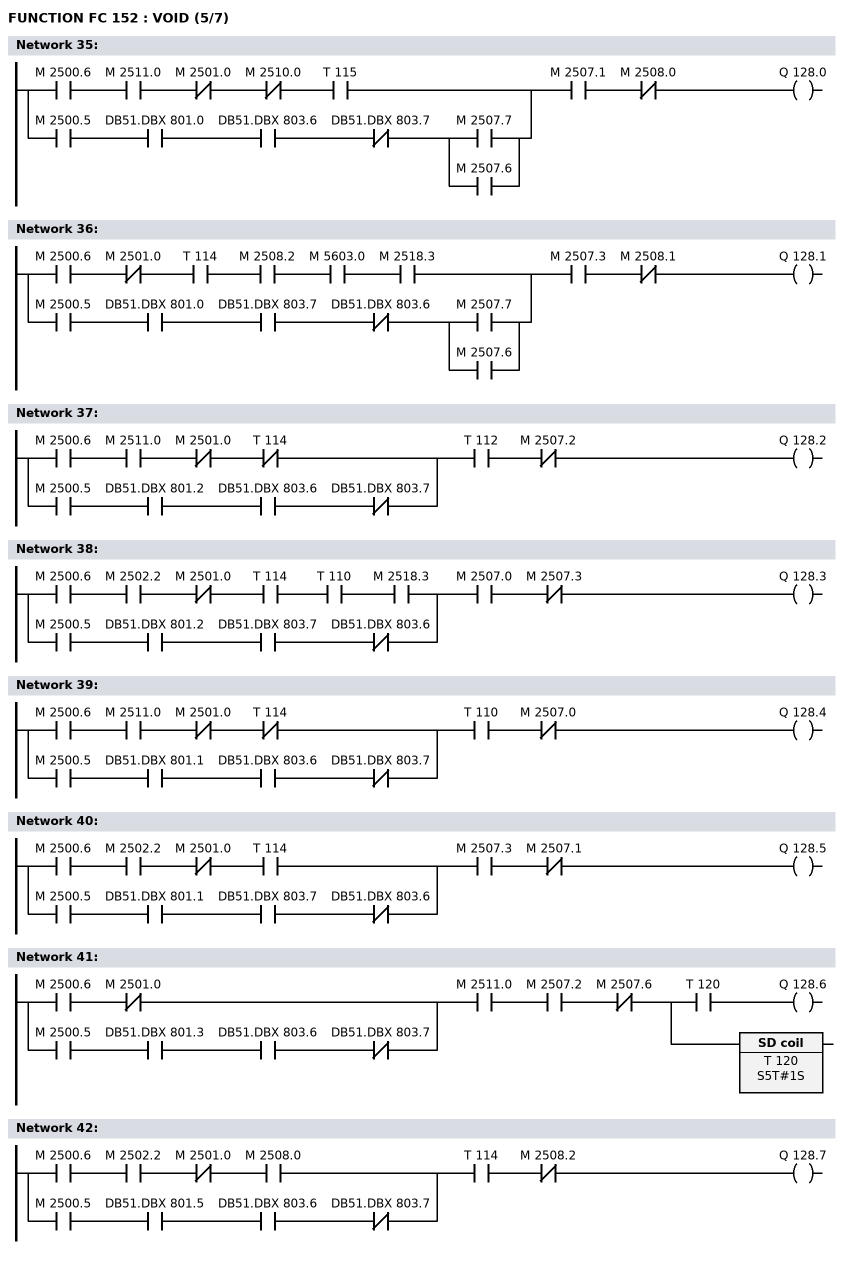

      A(    ;
      A     M   2500.6;
      A     M   2511.0;
      AN    M   2501.0;
      AN    M   2510.0;
      A     T    115;
      O     ;
      A     M   2500.5;
      A     DB51.DBX  801.0;
      A     DB51.DBX  803.6;
      AN    DB51.DBX  803.7;
      A(    ;
      O     M   2507.7;
      O     M   2507.6;
      )     ;
      )     ;
      A     M   2507.1;
      AN    M   2508.0;
      =     Q    128.0;
NETWORK
TITLE =

      A(    ;
      A     M   2500.6;
      AN    M   2501.0;
      A     T    114;
      A     M   2508.2;
      A     M   5603.0;
      A     M   2518.3;
      O     ;
      A     M   2500.5;
      A     DB51.DBX  801.0;
      A     DB51.DBX  803.7;
      AN    DB51.DBX  803.6;
      A(    ;
      O     M   2507.7;
      O     M   2507.6;
      )     ;
      )     ;
      A     M   2507.3;
      AN    M   2508.1;
      =     Q    128.1;
NETWORK
TITLE =

      A(    ;
      A     M   2500.6;
      A     M   2511.0;
      AN    M   2501.0;
      AN    T    114;
      O     ;
      A     M   2500.5;
      A     DB51.DBX  801.2;
      A     DB51.DBX  803.6;
      AN    DB51.DBX  803.7;
      )     ;
      A     T    112;
      AN    M   2507.2;
      =     Q    128.2;
NETWORK
TITLE =

      A(    ;
      A     M   2500.6;
      A     M   2502.2;
      AN    M   2501.0;
      A     T    114;
      A     T    110;
      A     M   2518.3;
      O     ;
      A     M   2500.5;
      A     DB51.DBX  801.2;
      A     DB51.DBX  803.7;
      AN    DB51.DBX  803.6;
      )     ;
      A     M   2507.0;
      AN    M   2507.3;
      =     Q    128.3;
NETWORK
TITLE =

      A(    ;
      A     M   2500.6;
      A     M   2511.0;
      AN    M   2501.0;
      AN    T    114;
      O     ;
      A     M   2500.5;
      A     DB51.DBX  801.1;
      A     DB51.DBX  803.6;
      AN    DB51.DBX  803.7;
      )     ;
      A     T    110;
      AN    M   2507.0;
      =     Q    128.4;
NETWORK
TITLE =

      A(    ;
      A     M   2500.6;
      A     M   2502.2;
      AN    M   2501.0;
      A     T    114;
      O     ;
      A     M   2500.5;
      A     DB51.DBX  801.1;
      A     DB51.DBX  803.7;
      AN    DB51.DBX  803.6;
      )     ;
      A     M   2507.3;
      AN    M   2507.1;
      =     Q    128.5;
NETWORK
TITLE =

      A(    ;
      A     M   2500.6;
      AN    M   2501.0;
      O     ;
      A     M   2500.5;
      A     DB51.DBX  801.3;
      A     DB51.DBX  803.6;
      AN    DB51.DBX  803.7;
      )     ;
      A     M   2511.0;
      A     M   2507.2;
      AN    M   2507.6;
      =     L      0.0;
      A     L      0.0;
      A     T    120;
      =     Q    128.6;
      A     L      0.0;
      BLD   102;
      L     S5T#1S;
      SD    T    120;
NETWORK
TITLE =

      A(    ;
      A     M   2500.6;
      A     M   2502.2;
      AN    M   2501.0;
      A     M   2508.0;
      O     ;
      A     M   2500.5;
      A     DB51.DBX  801.5;
      A     DB51.DBX  803.6;
      AN    DB51.DBX  803.7;
      )     ;
      A     T    114;
      AN    M   2508.2;
      =     Q    128.7;
NETWORK
TITLE =
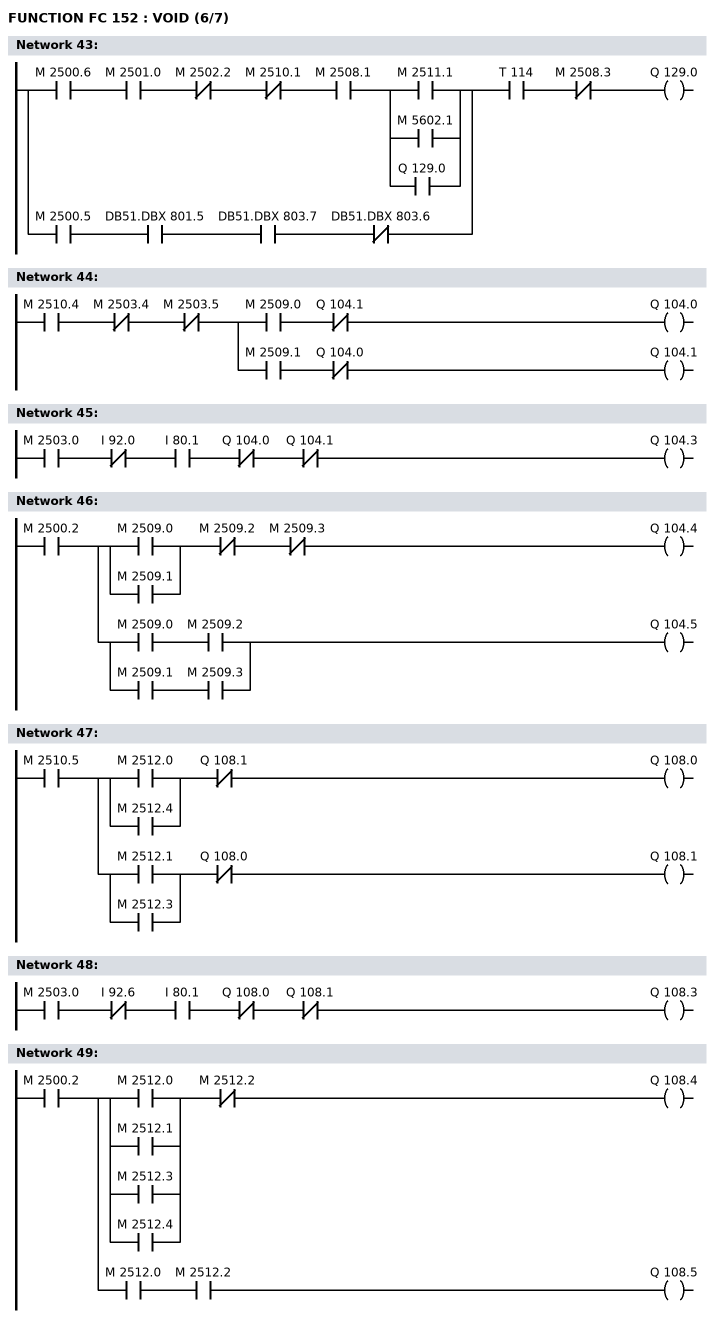

      A(    ;
      A     M   2500.6;
      A     M   2501.0;
      AN    M   2502.2;
      AN    M   2510.1;
      A     M   2508.1;
      A(    ;
      O     M   2511.1;
      O     M   5602.1;
      O     Q    129.0;
      )     ;
      O     ;
      A     M   2500.5;
      A     DB51.DBX  801.5;
      A     DB51.DBX  803.7;
      AN    DB51.DBX  803.6;
      )     ;
      A     T    114;
      AN    M   2508.3;
      =     Q    129.0;
NETWORK
TITLE =

      A     M   2510.4;
      AN    M   2503.4;
      AN    M   2503.5;
      =     L      0.0;
      A     L      0.0;
      A     M   2509.0;
      AN    Q    104.1;
      =     Q    104.0;
      A     L      0.0;
      A     M   2509.1;
      AN    Q    104.0;
      =     Q    104.1;
NETWORK
TITLE =

      A     M   2503.0;
      AN    I     92.0;
      A     I     80.1;
      AN    Q    104.0;
      AN    Q    104.1;
      =     Q    104.3;
NETWORK
TITLE =

      A     M   2500.2;
      =     L      0.0;
      A     L      0.0;
      A(    ;
      O     M   2509.0;
      O     M   2509.1;
      )     ;
      AN    M   2509.2;
      AN    M   2509.3;
      =     Q    104.4;
      A     L      0.0;
      A(    ;
      A     M   2509.0;
      A     M   2509.2;
      O     ;
      A     M   2509.1;
      A     M   2509.3;
      )     ;
      =     Q    104.5;
NETWORK
TITLE =

      A     M   2510.5;
      =     L      0.0;
      A     L      0.0;
      A(    ;
      O     M   2512.0;
      O     M   2512.4;
      )     ;
      AN    Q    108.1;
      =     Q    108.0;
      A     L      0.0;
      A(    ;
      O     M   2512.1;
      O     M   2512.3;
      )     ;
      AN    Q    108.0;
      =     Q    108.1;
NETWORK
TITLE =

      A     M   2503.0;
      AN    I     92.6;
      A     I     80.1;
      AN    Q    108.0;
      AN    Q    108.1;
      =     Q    108.3;
NETWORK
TITLE =

      A     M   2500.2;
      =     L      0.0;
      A     L      0.0;
      A(    ;
      O     M   2512.0;
      O     M   2512.1;
      O     M   2512.3;
      O     M   2512.4;
      )     ;
      AN    M   2512.2;
      =     Q    108.4;
      A     L      0.0;
      A     M   2512.0;
      A     M   2512.2;
      =     Q    108.5;
NETWORK
TITLE =
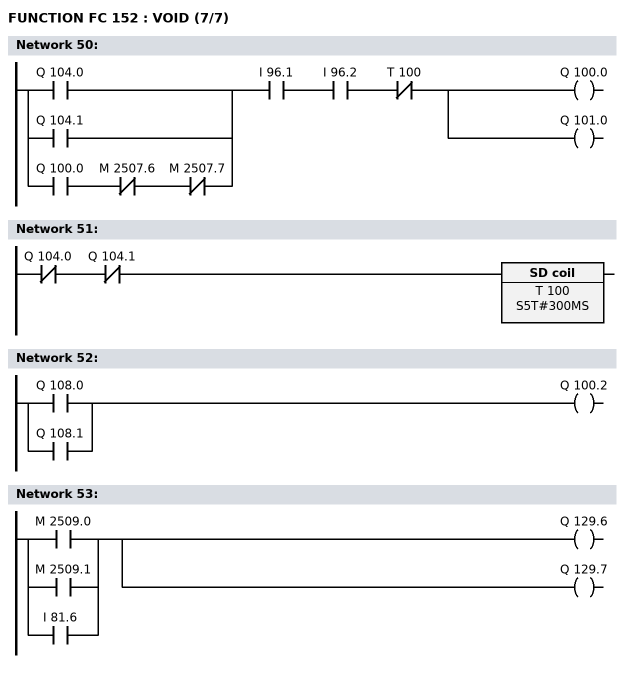

      A(    ;
      O     Q    104.0;
      O     Q    104.1;
      O     ;
      A     Q    100.0;
      AN    M   2507.6;
      AN    M   2507.7;
      )     ;
      A     I     96.1;
      A     I     96.2;
      AN    T    100;
      =     Q    100.0;
      =     Q    101.0;
NETWORK
TITLE =

      AN    Q    104.0;
      AN    Q    104.1;
      L     S5T#300MS;
      SD    T    100;
NETWORK
TITLE =

      O     Q    108.0;
      O     Q    108.1;
      =     Q    100.2;
NETWORK
TITLE =

      O     M   2509.0;
      O     M   2509.1;
      O     I     81.6;
      =     Q    129.6;
      =     Q    129.7;
END_FUNCTION

FUNCTION FC 159 : VOID
TITLE =
VERSION : 0.1

BEGIN
NETWORK
TITLE =
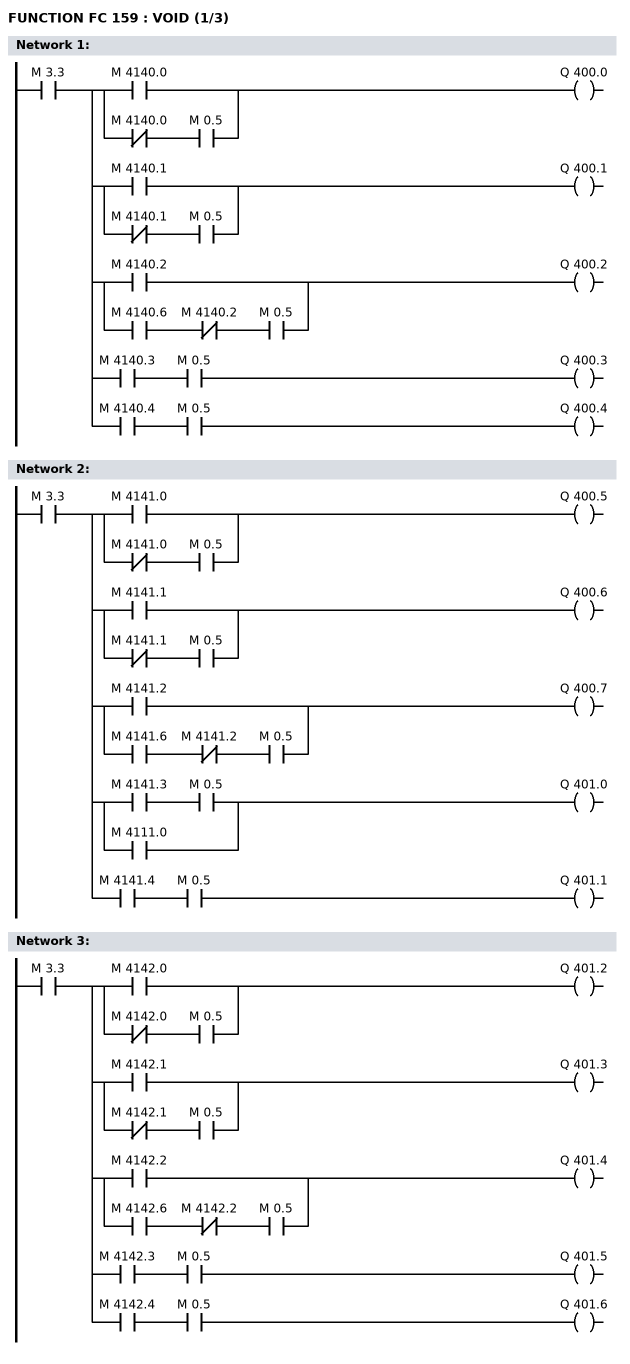

      A     M      3.3;
      =     L      0.0;
      A     L      0.0;
      A(    ;
      O     M   4140.0;
      O     ;
      AN    M   4140.0;
      A     M      0.5;
      )     ;
      =     Q    400.0;
      A     L      0.0;
      A(    ;
      O     M   4140.1;
      O     ;
      AN    M   4140.1;
      A     M      0.5;
      )     ;
      =     Q    400.1;
      A     L      0.0;
      A(    ;
      O     M   4140.2;
      O     ;
      A     M   4140.6;
      AN    M   4140.2;
      A     M      0.5;
      )     ;
      =     Q    400.2;
      A     L      0.0;
      A     M   4140.3;
      A     M      0.5;
      =     Q    400.3;
      A     L      0.0;
      A     M   4140.4;
      A     M      0.5;
      =     Q    400.4;
NETWORK
TITLE =

      A     M      3.3;
      =     L      0.0;
      A     L      0.0;
      A(    ;
      O     M   4141.0;
      O     ;
      AN    M   4141.0;
      A     M      0.5;
      )     ;
      =     Q    400.5;
      A     L      0.0;
      A(    ;
      O     M   4141.1;
      O     ;
      AN    M   4141.1;
      A     M      0.5;
      )     ;
      =     Q    400.6;
      A     L      0.0;
      A(    ;
      O     M   4141.2;
      O     ;
      A     M   4141.6;
      AN    M   4141.2;
      A     M      0.5;
      )     ;
      =     Q    400.7;
      A     L      0.0;
      A(    ;
      A     M   4141.3;
      A     M      0.5;
      O     M   4111.0;
      )     ;
      =     Q    401.0;
      A     L      0.0;
      A     M   4141.4;
      A     M      0.5;
      =     Q    401.1;
NETWORK
TITLE =

      A     M      3.3;
      =     L      0.0;
      A     L      0.0;
      A(    ;
      O     M   4142.0;
      O     ;
      AN    M   4142.0;
      A     M      0.5;
      )     ;
      =     Q    401.2;
      A     L      0.0;
      A(    ;
      O     M   4142.1;
      O     ;
      AN    M   4142.1;
      A     M      0.5;
      )     ;
      =     Q    401.3;
      A     L      0.0;
      A(    ;
      O     M   4142.2;
      O     ;
      A     M   4142.6;
      AN    M   4142.2;
      A     M      0.5;
      )     ;
      =     Q    401.4;
      A     L      0.0;
      A     M   4142.3;
      A     M      0.5;
      =     Q    401.5;
      A     L      0.0;
      A     M   4142.4;
      A     M      0.5;
      =     Q    401.6;
NETWORK
TITLE =
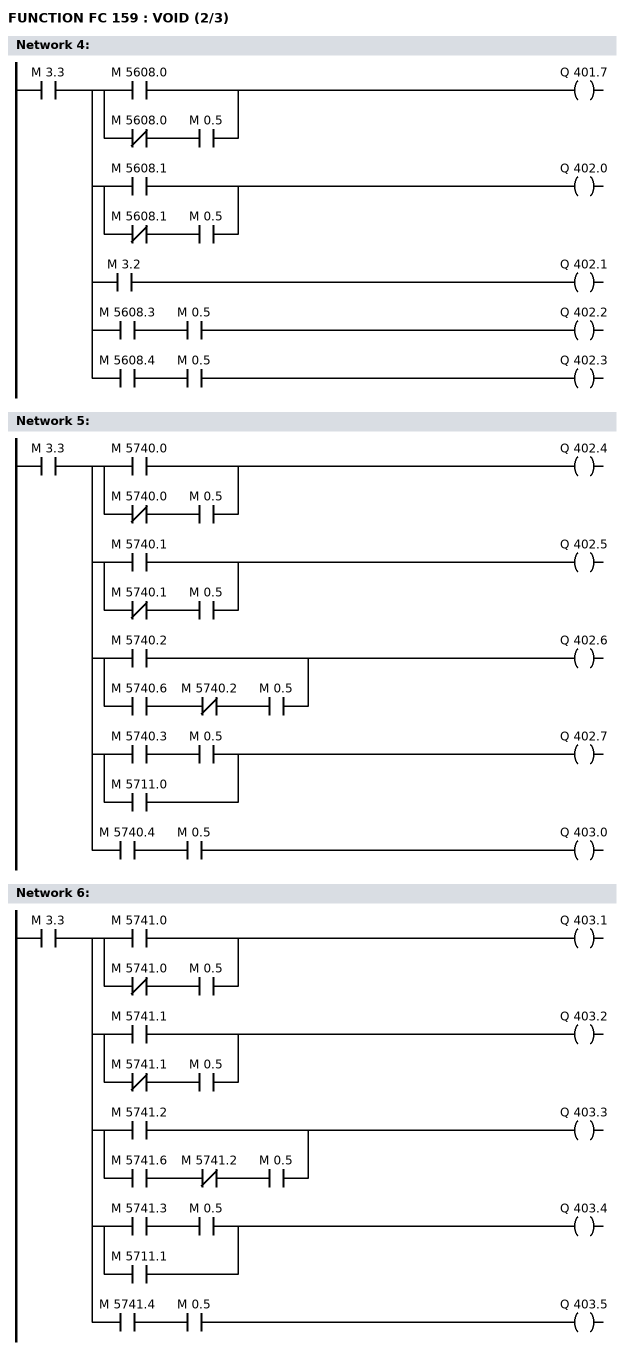

      A     M      3.3;
      =     L      0.0;
      A     L      0.0;
      A(    ;
      O     M   5608.0;
      O     ;
      AN    M   5608.0;
      A     M      0.5;
      )     ;
      =     Q    401.7;
      A     L      0.0;
      A(    ;
      O     M   5608.1;
      O     ;
      AN    M   5608.1;
      A     M      0.5;
      )     ;
      =     Q    402.0;
      A     L      0.0;
      A     M      3.2;
      =     Q    402.1;
      A     L      0.0;
      A     M   5608.3;
      A     M      0.5;
      =     Q    402.2;
      A     L      0.0;
      A     M   5608.4;
      A     M      0.5;
      =     Q    402.3;
NETWORK
TITLE =

      A     M      3.3;
      =     L      0.0;
      A     L      0.0;
      A(    ;
      O     M   5740.0;
      O     ;
      AN    M   5740.0;
      A     M      0.5;
      )     ;
      =     Q    402.4;
      A     L      0.0;
      A(    ;
      O     M   5740.1;
      O     ;
      AN    M   5740.1;
      A     M      0.5;
      )     ;
      =     Q    402.5;
      A     L      0.0;
      A(    ;
      O     M   5740.2;
      O     ;
      A     M   5740.6;
      AN    M   5740.2;
      A     M      0.5;
      )     ;
      =     Q    402.6;
      A     L      0.0;
      A(    ;
      A     M   5740.3;
      A     M      0.5;
      O     M   5711.0;
      )     ;
      =     Q    402.7;
      A     L      0.0;
      A     M   5740.4;
      A     M      0.5;
      =     Q    403.0;
NETWORK
TITLE =

      A     M      3.3;
      =     L      0.0;
      A     L      0.0;
      A(    ;
      O     M   5741.0;
      O     ;
      AN    M   5741.0;
      A     M      0.5;
      )     ;
      =     Q    403.1;
      A     L      0.0;
      A(    ;
      O     M   5741.1;
      O     ;
      AN    M   5741.1;
      A     M      0.5;
      )     ;
      =     Q    403.2;
      A     L      0.0;
      A(    ;
      O     M   5741.2;
      O     ;
      A     M   5741.6;
      AN    M   5741.2;
      A     M      0.5;
      )     ;
      =     Q    403.3;
      A     L      0.0;
      A(    ;
      A     M   5741.3;
      A     M      0.5;
      O     M   5711.1;
      )     ;
      =     Q    403.4;
      A     L      0.0;
      A     M   5741.4;
      A     M      0.5;
      =     Q    403.5;
NETWORK
TITLE =
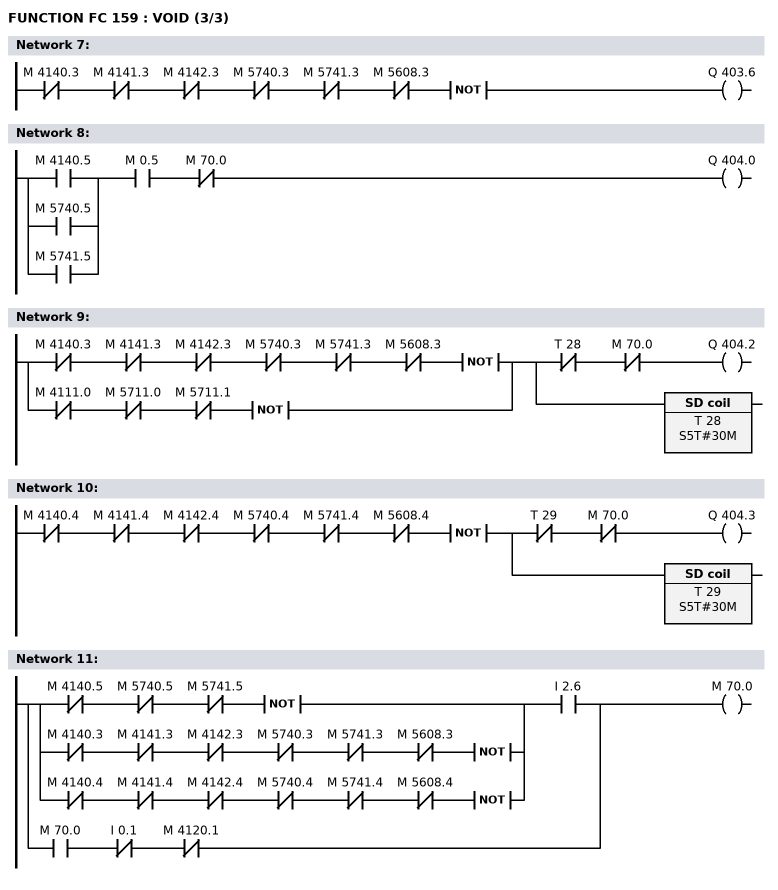

      AN    M   4140.3;
      AN    M   4141.3;
      AN    M   4142.3;
      AN    M   5740.3;
      AN    M   5741.3;
      AN    M   5608.3;
      NOT   ;
      =     Q    403.6;
NETWORK
TITLE =

      A(    ;
      O     M   4140.5;
      O     M   5740.5;
      O     M   5741.5;
      )     ;
      A     M      0.5;
      AN    M     70.0;
      =     Q    404.0;
NETWORK
TITLE =

      AN    M   4140.3;
      AN    M   4141.3;
      AN    M   4142.3;
      AN    M   5740.3;
      AN    M   5741.3;
      AN    M   5608.3;
      NOT   ;
      O(    ;
      AN    M   4111.0;
      AN    M   5711.0;
      AN    M   5711.1;
      NOT   ;
      )     ;
      =     L      0.0;
      A     L      0.0;
      AN    T     28;
      AN    M     70.0;
      =     Q    404.2;
      A     L      0.0;
      BLD   102;
      L     S5T#30M;
      SD    T     28;
NETWORK
TITLE =

      AN    M   4140.4;
      AN    M   4141.4;
      AN    M   4142.4;
      AN    M   5740.4;
      AN    M   5741.4;
      AN    M   5608.4;
      NOT   ;
      =     L      0.0;
      A     L      0.0;
      AN    T     29;
      AN    M     70.0;
      =     Q    404.3;
      A     L      0.0;
      BLD   102;
      L     S5T#30M;
      SD    T     29;
NETWORK
TITLE =

      A(    ;
      AN    M   4140.5;
      AN    M   5740.5;
      AN    M   5741.5;
      NOT   ;
      O(    ;
      AN    M   4140.3;
      AN    M   4141.3;
      AN    M   4142.3;
      AN    M   5740.3;
      AN    M   5741.3;
      AN    M   5608.3;
      NOT   ;
      )     ;
      O(    ;
      AN    M   4140.4;
      AN    M   4141.4;
      AN    M   4142.4;
      AN    M   5740.4;
      AN    M   5741.4;
      AN    M   5608.4;
      NOT   ;
      )     ;
      )     ;
      A     I      2.6;
      O     ;
      A     M     70.0;
      AN    I      0.1;
      AN    M   4120.1;
      =     M     70.0;
END_FUNCTION

FUNCTION FC 324 : VOID
TITLE =
VERSION : 0.1

BEGIN
NETWORK
TITLE =DP DIAGNOSTIC FOR DP MASTER SYSTEM(1)

      AN    OV;
      =     L      0.0;
      BLD   103;
      A     OV;
      =     L      0.1;
      BLD   103;
      CALL FC   325 (
           CHECK_ACTIV              := L      0.0,
           EXTERNAL_DP_INTERFACE    := L      0.1,
           DP_MASTERSYSTEM          := 1,
           DATA_FIELD               := P#DB325.DBX0.0 BYTE 50,
           SUM_SLAVES_DIAG          := DB325.DBW   82,
           LIST_SLAVES_NOT_PRESENT  := P#DB325.DBX 50.0 DWORD 4,
           LIST_SLAVES_ERROR        := P#DB325.DBX 66.0 DWORD 4,
           RETVAL                   := DB325.DBW   84,
           BUSY                     := DB325.DBX   90.0);
      NOP   0;
NETWORK
TITLE =705R1
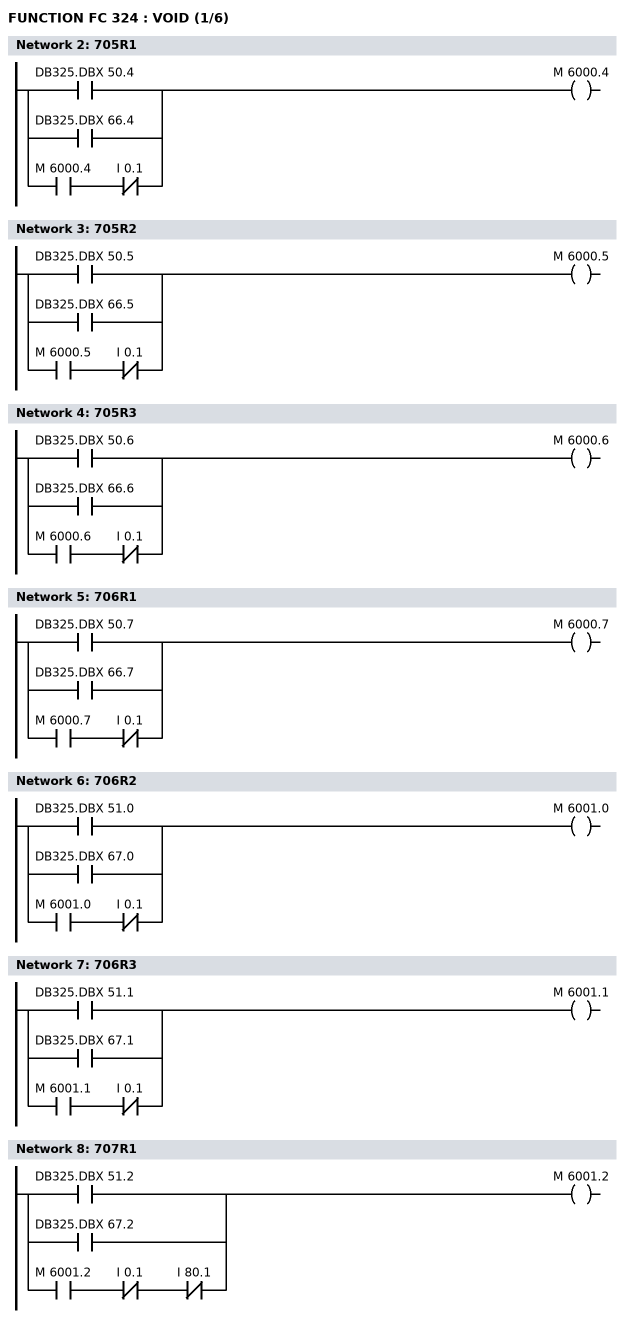

      O     DB325.DBX   50.4;
      O     DB325.DBX   66.4;
      O     ;
      A     M   6000.4;
      AN    I      0.1;
      =     M   6000.4;
NETWORK
TITLE =705R2

      O     DB325.DBX   50.5;
      O     DB325.DBX   66.5;
      O     ;
      A     M   6000.5;
      AN    I      0.1;
      =     M   6000.5;
NETWORK
TITLE =705R3

      O     DB325.DBX   50.6;
      O     DB325.DBX   66.6;
      O     ;
      A     M   6000.6;
      AN    I      0.1;
      =     M   6000.6;
NETWORK
TITLE =706R1

      O     DB325.DBX   50.7;
      O     DB325.DBX   66.7;
      O     ;
      A     M   6000.7;
      AN    I      0.1;
      =     M   6000.7;
NETWORK
TITLE =706R2

      O     DB325.DBX   51.0;
      O     DB325.DBX   67.0;
      O     ;
      A     M   6001.0;
      AN    I      0.1;
      =     M   6001.0;
NETWORK
TITLE =706R3

      O     DB325.DBX   51.1;
      O     DB325.DBX   67.1;
      O     ;
      A     M   6001.1;
      AN    I      0.1;
      =     M   6001.1;
NETWORK
TITLE =707R1

      O     DB325.DBX   51.2;
      O     DB325.DBX   67.2;
      O     ;
      A     M   6001.2;
      AN    I      0.1;
      AN    I     80.1;
      =     M   6001.2;
NETWORK
TITLE =707R2
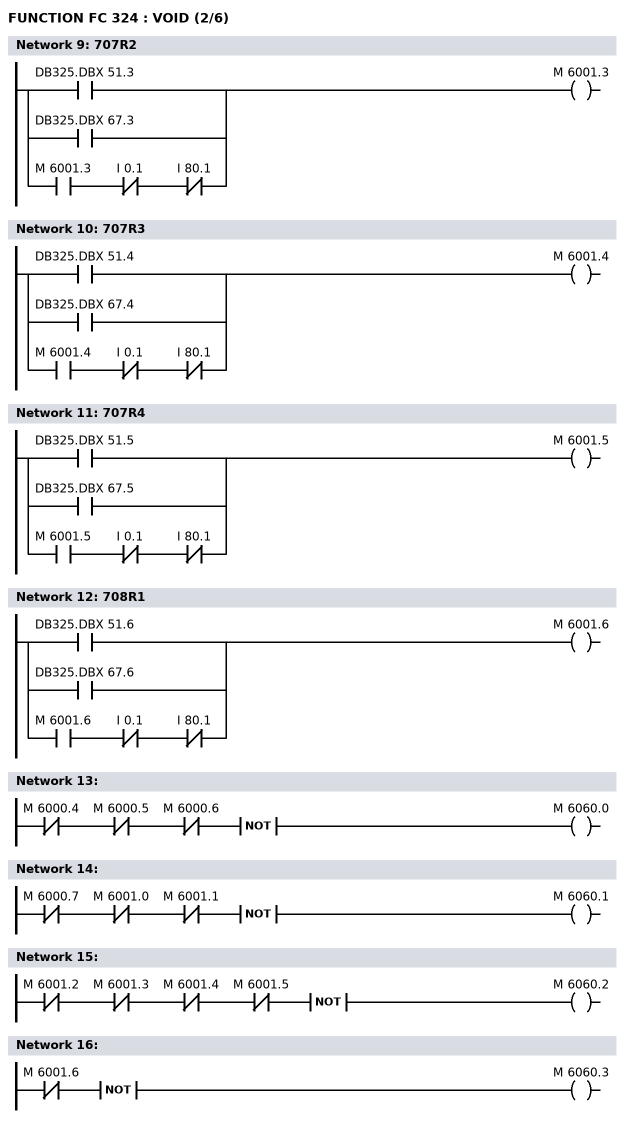

      O     DB325.DBX   51.3;
      O     DB325.DBX   67.3;
      O     ;
      A     M   6001.3;
      AN    I      0.1;
      AN    I     80.1;
      =     M   6001.3;
NETWORK
TITLE =707R3

      O     DB325.DBX   51.4;
      O     DB325.DBX   67.4;
      O     ;
      A     M   6001.4;
      AN    I      0.1;
      AN    I     80.1;
      =     M   6001.4;
NETWORK
TITLE =707R4

      O     DB325.DBX   51.5;
      O     DB325.DBX   67.5;
      O     ;
      A     M   6001.5;
      AN    I      0.1;
      AN    I     80.1;
      =     M   6001.5;
NETWORK
TITLE =708R1

      O     DB325.DBX   51.6;
      O     DB325.DBX   67.6;
      O     ;
      A     M   6001.6;
      AN    I      0.1;
      AN    I     80.1;
      =     M   6001.6;
NETWORK
TITLE =

      AN    M   6000.4;
      AN    M   6000.5;
      AN    M   6000.6;
      NOT   ;
      =     M   6060.0;
NETWORK
TITLE =

      AN    M   6000.7;
      AN    M   6001.0;
      AN    M   6001.1;
      NOT   ;
      =     M   6060.1;
NETWORK
TITLE =

      AN    M   6001.2;
      AN    M   6001.3;
      AN    M   6001.4;
      AN    M   6001.5;
      NOT   ;
      =     M   6060.2;
NETWORK
TITLE =

      AN    M   6001.6;
      NOT   ;
      =     M   6060.3;
NETWORK
TITLE =
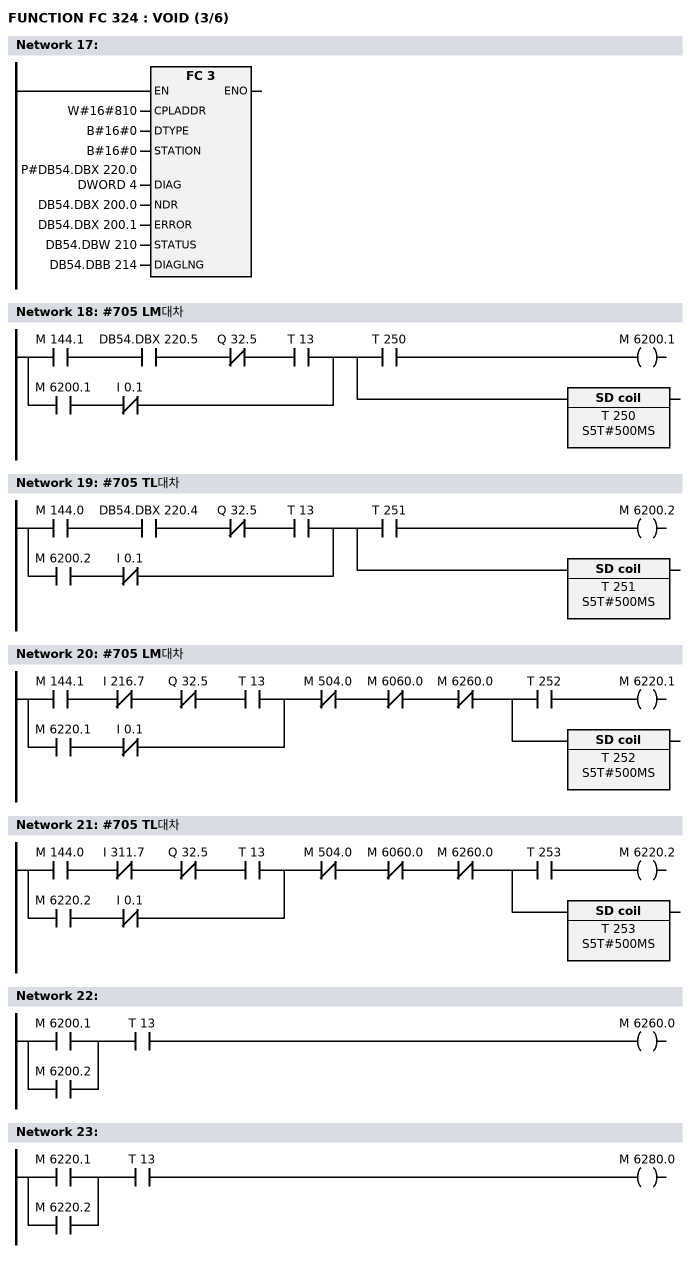

      CALL FC     3 (
           CPLADDR                  := W#16#810,
           DTYPE                    := B#16#0,
           STATION                  := B#16#0,
           DIAG                     := P#DB54.DBX 220.0 DWORD 4,
           NDR                      := DB54.DBX  200.0,
           ERROR                    := DB54.DBX  200.1,
           STATUS                   := DB54.DBW  210,
           DIAGLNG                  := DB54.DBB  214);
      NOP   0;
NETWORK
TITLE =#705 LM대차

      A     M    144.1;
      A     DB54.DBX  220.5;
      AN    Q     32.5;
      A     T     13;
      O     ;
      A     M   6200.1;
      AN    I      0.1;
      =     L      0.0;
      A     L      0.0;
      A     T    250;
      =     M   6200.1;
      A     L      0.0;
      BLD   102;
      L     S5T#500MS;
      SD    T    250;
NETWORK
TITLE =#705 TL대차

      A     M    144.0;
      A     DB54.DBX  220.4;
      AN    Q     32.5;
      A     T     13;
      O     ;
      A     M   6200.2;
      AN    I      0.1;
      =     L      0.0;
      A     L      0.0;
      A     T    251;
      =     M   6200.2;
      A     L      0.0;
      BLD   102;
      L     S5T#500MS;
      SD    T    251;
NETWORK
TITLE =#705 LM대차

      A(    ;
      A     M    144.1;
      AN    I    216.7;
      AN    Q     32.5;
      A     T     13;
      O     ;
      A     M   6220.1;
      AN    I      0.1;
      )     ;
      AN    M    504.0;
      AN    M   6060.0;
      AN    M   6260.0;
      =     L      0.0;
      A     L      0.0;
      A     T    252;
      =     M   6220.1;
      A     L      0.0;
      BLD   102;
      L     S5T#500MS;
      SD    T    252;
NETWORK
TITLE =#705 TL대차

      A(    ;
      A     M    144.0;
      AN    I    311.7;
      AN    Q     32.5;
      A     T     13;
      O     ;
      A     M   6220.2;
      AN    I      0.1;
      )     ;
      AN    M    504.0;
      AN    M   6060.0;
      AN    M   6260.0;
      =     L      0.0;
      A     L      0.0;
      A     T    253;
      =     M   6220.2;
      A     L      0.0;
      BLD   102;
      L     S5T#500MS;
      SD    T    253;
NETWORK
TITLE =

      A(    ;
      O     M   6200.1;
      O     M   6200.2;
      )     ;
      A     T     13;
      =     M   6260.0;
NETWORK
TITLE =

      A(    ;
      O     M   6220.1;
      O     M   6220.2;
      )     ;
      A     T     13;
      =     M   6280.0;
NETWORK
TITLE =
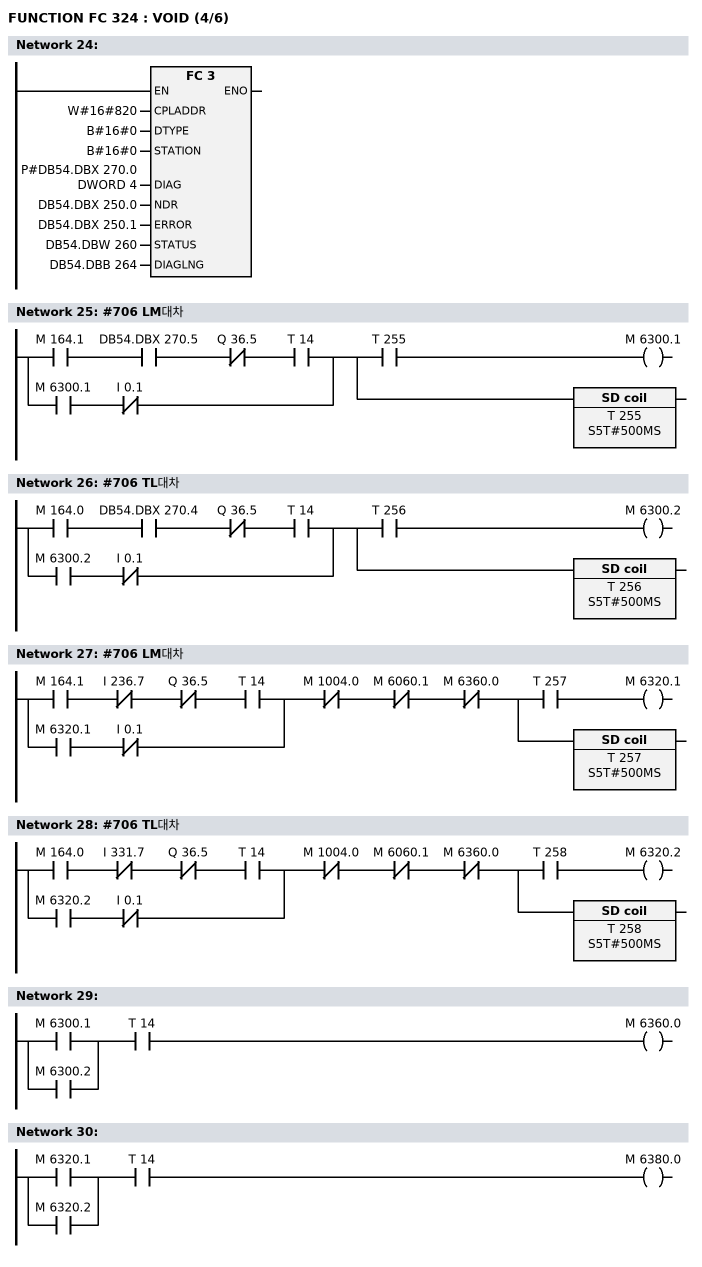

      CALL FC     3 (
           CPLADDR                  := W#16#820,
           DTYPE                    := B#16#0,
           STATION                  := B#16#0,
           DIAG                     := P#DB54.DBX 270.0 DWORD 4,
           NDR                      := DB54.DBX  250.0,
           ERROR                    := DB54.DBX  250.1,
           STATUS                   := DB54.DBW  260,
           DIAGLNG                  := DB54.DBB  264);
      NOP   0;
NETWORK
TITLE =#706 LM대차

      A     M    164.1;
      A     DB54.DBX  270.5;
      AN    Q     36.5;
      A     T     14;
      O     ;
      A     M   6300.1;
      AN    I      0.1;
      =     L      0.0;
      A     L      0.0;
      A     T    255;
      =     M   6300.1;
      A     L      0.0;
      BLD   102;
      L     S5T#500MS;
      SD    T    255;
NETWORK
TITLE =#706 TL대차

      A     M    164.0;
      A     DB54.DBX  270.4;
      AN    Q     36.5;
      A     T     14;
      O     ;
      A     M   6300.2;
      AN    I      0.1;
      =     L      0.0;
      A     L      0.0;
      A     T    256;
      =     M   6300.2;
      A     L      0.0;
      BLD   102;
      L     S5T#500MS;
      SD    T    256;
NETWORK
TITLE =#706 LM대차

      A(    ;
      A     M    164.1;
      AN    I    236.7;
      AN    Q     36.5;
      A     T     14;
      O     ;
      A     M   6320.1;
      AN    I      0.1;
      )     ;
      AN    M   1004.0;
      AN    M   6060.1;
      AN    M   6360.0;
      =     L      0.0;
      A     L      0.0;
      A     T    257;
      =     M   6320.1;
      A     L      0.0;
      BLD   102;
      L     S5T#500MS;
      SD    T    257;
NETWORK
TITLE =#706 TL대차

      A(    ;
      A     M    164.0;
      AN    I    331.7;
      AN    Q     36.5;
      A     T     14;
      O     ;
      A     M   6320.2;
      AN    I      0.1;
      )     ;
      AN    M   1004.0;
      AN    M   6060.1;
      AN    M   6360.0;
      =     L      0.0;
      A     L      0.0;
      A     T    258;
      =     M   6320.2;
      A     L      0.0;
      BLD   102;
      L     S5T#500MS;
      SD    T    258;
NETWORK
TITLE =

      A(    ;
      O     M   6300.1;
      O     M   6300.2;
      )     ;
      A     T     14;
      =     M   6360.0;
NETWORK
TITLE =

      A(    ;
      O     M   6320.1;
      O     M   6320.2;
      )     ;
      A     T     14;
      =     M   6380.0;
NETWORK
TITLE =
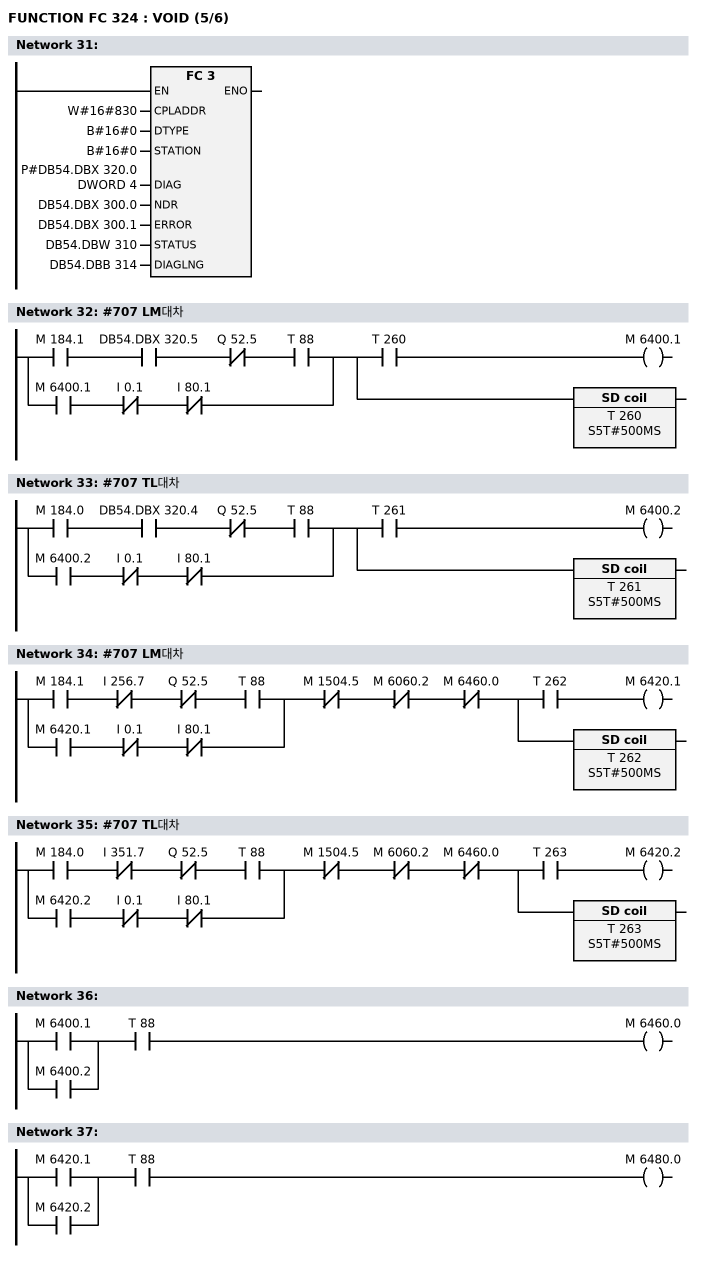

      CALL FC     3 (
           CPLADDR                  := W#16#830,
           DTYPE                    := B#16#0,
           STATION                  := B#16#0,
           DIAG                     := P#DB54.DBX 320.0 DWORD 4,
           NDR                      := DB54.DBX  300.0,
           ERROR                    := DB54.DBX  300.1,
           STATUS                   := DB54.DBW  310,
           DIAGLNG                  := DB54.DBB  314);
      NOP   0;
NETWORK
TITLE =#707 LM대차

      A     M    184.1;
      A     DB54.DBX  320.5;
      AN    Q     52.5;
      A     T     88;
      O     ;
      A     M   6400.1;
      AN    I      0.1;
      AN    I     80.1;
      =     L      0.0;
      A     L      0.0;
      A     T    260;
      =     M   6400.1;
      A     L      0.0;
      BLD   102;
      L     S5T#500MS;
      SD    T    260;
NETWORK
TITLE =#707 TL대차

      A     M    184.0;
      A     DB54.DBX  320.4;
      AN    Q     52.5;
      A     T     88;
      O     ;
      A     M   6400.2;
      AN    I      0.1;
      AN    I     80.1;
      =     L      0.0;
      A     L      0.0;
      A     T    261;
      =     M   6400.2;
      A     L      0.0;
      BLD   102;
      L     S5T#500MS;
      SD    T    261;
NETWORK
TITLE =#707 LM대차

      A(    ;
      A     M    184.1;
      AN    I    256.7;
      AN    Q     52.5;
      A     T     88;
      O     ;
      A     M   6420.1;
      AN    I      0.1;
      AN    I     80.1;
      )     ;
      AN    M   1504.5;
      AN    M   6060.2;
      AN    M   6460.0;
      =     L      0.0;
      A     L      0.0;
      A     T    262;
      =     M   6420.1;
      A     L      0.0;
      BLD   102;
      L     S5T#500MS;
      SD    T    262;
NETWORK
TITLE =#707 TL대차

      A(    ;
      A     M    184.0;
      AN    I    351.7;
      AN    Q     52.5;
      A     T     88;
      O     ;
      A     M   6420.2;
      AN    I      0.1;
      AN    I     80.1;
      )     ;
      AN    M   1504.5;
      AN    M   6060.2;
      AN    M   6460.0;
      =     L      0.0;
      A     L      0.0;
      A     T    263;
      =     M   6420.2;
      A     L      0.0;
      BLD   102;
      L     S5T#500MS;
      SD    T    263;
NETWORK
TITLE =

      A(    ;
      O     M   6400.1;
      O     M   6400.2;
      )     ;
      A     T     88;
      =     M   6460.0;
NETWORK
TITLE =

      A(    ;
      O     M   6420.1;
      O     M   6420.2;
      )     ;
      A     T     88;
      =     M   6480.0;
NETWORK
TITLE =
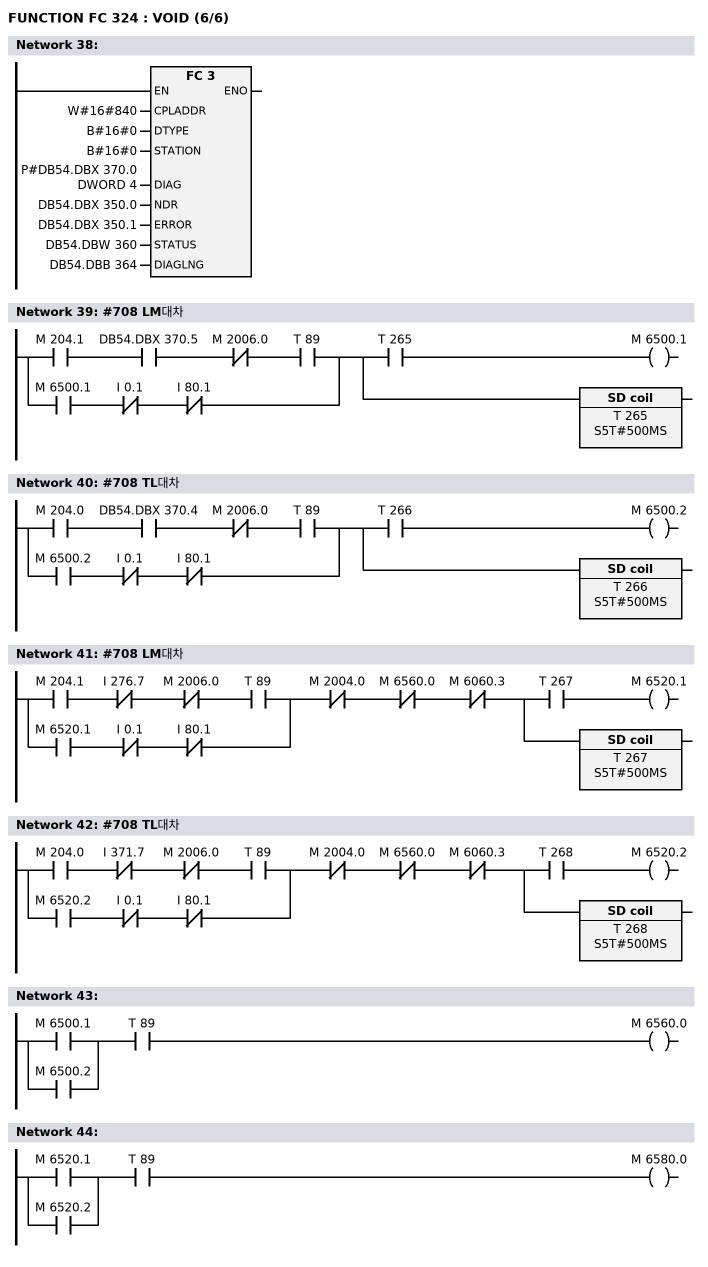

      CALL FC     3 (
           CPLADDR                  := W#16#840,
           DTYPE                    := B#16#0,
           STATION                  := B#16#0,
           DIAG                     := P#DB54.DBX 370.0 DWORD 4,
           NDR                      := DB54.DBX  350.0,
           ERROR                    := DB54.DBX  350.1,
           STATUS                   := DB54.DBW  360,
           DIAGLNG                  := DB54.DBB  364);
      NOP   0;
NETWORK
TITLE =#708 LM대차

      A     M    204.1;
      A     DB54.DBX  370.5;
      AN    M   2006.0;
      A     T     89;
      O     ;
      A     M   6500.1;
      AN    I      0.1;
      AN    I     80.1;
      =     L      0.0;
      A     L      0.0;
      A     T    265;
      =     M   6500.1;
      A     L      0.0;
      BLD   102;
      L     S5T#500MS;
      SD    T    265;
NETWORK
TITLE =#708 TL대차

      A     M    204.0;
      A     DB54.DBX  370.4;
      AN    M   2006.0;
      A     T     89;
      O     ;
      A     M   6500.2;
      AN    I      0.1;
      AN    I     80.1;
      =     L      0.0;
      A     L      0.0;
      A     T    266;
      =     M   6500.2;
      A     L      0.0;
      BLD   102;
      L     S5T#500MS;
      SD    T    266;
NETWORK
TITLE =#708 LM대차

      A(    ;
      A     M    204.1;
      AN    I    276.7;
      AN    M   2006.0;
      A     T     89;
      O     ;
      A     M   6520.1;
      AN    I      0.1;
      AN    I     80.1;
      )     ;
      AN    M   2004.0;
      AN    M   6560.0;
      AN    M   6060.3;
      =     L      0.0;
      A     L      0.0;
      A     T    267;
      =     M   6520.1;
      A     L      0.0;
      BLD   102;
      L     S5T#500MS;
      SD    T    267;
NETWORK
TITLE =#708 TL대차

      A(    ;
      A     M    204.0;
      AN    I    371.7;
      AN    M   2006.0;
      A     T     89;
      O     ;
      A     M   6520.2;
      AN    I      0.1;
      AN    I     80.1;
      )     ;
      AN    M   2004.0;
      AN    M   6560.0;
      AN    M   6060.3;
      =     L      0.0;
      A     L      0.0;
      A     T    268;
      =     M   6520.2;
      A     L      0.0;
      BLD   102;
      L     S5T#500MS;
      SD    T    268;
NETWORK
TITLE =

      A(    ;
      O     M   6500.1;
      O     M   6500.2;
      )     ;
      A     T     89;
      =     M   6560.0;
NETWORK
TITLE =

      A(    ;
      O     M   6520.1;
      O     M   6520.2;
      )     ;
      A     T     89;
      =     M   6580.0;
END_FUNCTION

FUNCTION_BLOCK FB 406
TITLE =Data Block Move Program
AUTHOR : HMC
FAMILY : Car_Type
NAME : Car_Type
VERSION : 1.0


VAR_INPUT
  FWD_Pulse : BOOL ;
  RET_Pulse : BOOL ;
  Source_DB : INT ;
  Start_Add : INT ;
  Stn_Amount : INT ;
  Byte_per_Stn : INT ;
  Cpu_Run_Pulse : BOOL ;
END_VAR
VAR_OUTPUT
  Complete : BOOL ;
END_VAR
VAR
  Operation : BOOL ;
  Mask_Arr : ARRAY  [0 .. 599 ] OF BYTE ;
  Ret : INT ;
  Data_Type : WORD ;
  Data_Length : INT ;
  Secend_Stn_Add : INT ;
  Fill_Source : WORD ;
END_VAR
VAR_TEMP
  First_Stn : ANY ;
  Mask : ANY ;
  Second_Stn : ANY ;
  Save_AR1 : DWORD ;
  Save_AR2 : DWORD ;
  Save_DB : INT ;
  Save_DI : INT ;
  First_Stn_1 : ANY ;
END_VAR
BEGIN
NETWORK
TITLE =Save adress register and DB's

      TAR1  #Save_AR1; // Save adress register 1
      TAR2  #Save_AR2; // Save adress register 2
      L     DBNO; // loads the number of the shared open data block
      T     #Save_DB;
      L     DINO; // loads the number of the opened instance data block
      T     #Save_DI;
NETWORK
TITLE =Operation Pulse

      O     #FWD_Pulse; // External ForwardOperation Signal
      O     #RET_Pulse; // External Return Operation Signal
      FP    #Operation; // Operation Pulse
      JNB   _End; // Jump to End
NETWORK
TITLE =Data Type Select In ANY Type Parameter

      A(    ; // If Source DB is Not Zero
      L     #Source_DB;
      L     0;
      <>I   ;
      )     ;
      JNB   _001; // Jump to Next Step
      L     W#16#8400; // Load "8400" _ Means "DB Area"
      T     #Data_Type; // Transfer to Data_Type
_001: NOP   0;
NETWORK
TITLE =Data Type Select In ANY Type Parameter

      A(    ; // If DB_NO is Zero
      L     #Source_DB;
      L     0;
      ==I   ;
      )     ;
      JNB   _002; // Jump to Next Step
      L     W#16#8300; // Load "8300" _ Means "Bit Memory Area"
      T     #Data_Type; // Transfer to Data_Type
_002: NOP   0;
NETWORK
TITLE =Data Length Select

      L     #Stn_Amount; // Station Amount - 1
      L     1;
      -I    ;
      L     #Byte_per_Stn; // Multi Length Per Station
      *I    ;
      T     #Data_Length; // Transfer to Data Length
NETWORK
TITLE =2nd Station Address Select

      L     #Start_Add; // Pluse Start Address And Length
      L     #Byte_per_Stn;
      +I    ;
      T     #Secend_Stn_Add; // Transfer to Second Station Address
NETWORK
TITLE =Make a "ANY" Type Data

      LAR1  P##First_Stn; // Load 1st Station Address of ANY Pointer In "AR1"

      L     B#16#10; // Load Syntax ID For S7 "10"
      T     LB [AR1,P#0.0]; // Transfer ID to the ANY Pointer

      L     B#16#2; // Load Data Type _ "2" means "BYTE"
      T     LB [AR1,P#1.0]; // Transfer Data Type to the ANY Pointer

      L     #Data_Length; // Load the Length of Source Data
      T     LW [AR1,P#2.0]; // Transfer the Numbers to the ANY Pointer

      L     #Source_DB; // Load DB Number _ "0" means don't use "DB"
      T     LW [AR1,P#4.0]; // Transfer the Numbers to the ANY Pointer

      L     #Data_Type; // Load Data Type _ "83" means "Bit Memory" Area
      T     LW [AR1,P#6.0]; //                  "84" means "DB" Area

      L     #Start_Add; // Load Start Address
      SLW   3; // Shift Left Word _ "3" Bit
      T     LW [AR1,P#8.0]; // Transfer the Address to the ANY Pointer

      LAR1  P##Mask; // Load 2nd Station Address of ANY Pointer In "AR1"

      L     B#16#10; //Load Syntax ID For S7 "10"
      T     LB [AR1,P#0.0]; //Load Syntax ID For S7 "10"

      L     B#16#2; //  Load Data Type _ "2" means "BYTE"
      T     LB [AR1,P#1.0]; // Transfer Data Type to the ANY Pointer

      L     #Data_Length; // Load the Length of Target Data
      T     LW [AR1,P#2.0]; // Transfer the Numbers to the ANY Pointer

      L     #Save_DI; // Load DB Number _ "0" means don't use "DB"
      T     LW [AR1,P#4.0]; // Transfer the Numbers to the ANY Pointer

      L     #Data_Type; // Load Data Type _ "83" means "Bit Memory" Area
      T     LW [AR1,P#6.0]; //                  "84" means "DB" Area

      L     16; //  Load Start Address
      SLW   3; // Shift Left Word _ "3" Bit
      T     LW [AR1,P#8.0]; // Transfer the Address to the ANY Pointer

NETWORK
TITLE =Make a "ANY" Type Data

      LAR1  P##Second_Stn; // Load 1st Station Address of ANY Pointer In "AR1"

      L     B#16#10; // Load Syntax ID For S7 "10"
      T     LB [AR1,P#0.0]; // Transfer ID to the ANY Pointer

      L     B#16#2; // Load Data Type _ "2" means "BYTE"
      T     LB [AR1,P#1.0]; // Transfer Data Type to the ANY Pointer

      L     #Data_Length; // Load the Length of Source Data
      T     LW [AR1,P#2.0]; // Transfer the Numbers to the ANY Pointer

      L     #Source_DB; // Load DB Number _ "0" means don't use "DB"
      T     LW [AR1,P#4.0]; // Transfer the Numbers to the ANY Pointer

      L     #Data_Type; // Load Data Type _ "83" means "Bit Memory" Area
      T     LW [AR1,P#6.0]; //                  "84" means "DB" Area

      L     #Secend_Stn_Add; // Load Second Station Address
      SLW   3; // Shift Left Word _ "3" Bit
      T     LW [AR1,P#8.0]; // Transfer the Address to the ANY Pointer
NETWORK
TITLE =Reset Car Type Transfer Complete Signal

      O     #FWD_Pulse; // External Forward Operation Signal
      O     #RET_Pulse; // External Return Operation Signal
      R     #Complete; // Reset Complete Signal
NETWORK
TITLE =Make Fill Source Data

      L     0;
      T     #Fill_Source;
NETWORK
TITLE =Fwd Block Move to Mask Area

      A     #FWD_Pulse; // External Forward Operation Signal
      AN    #Complete; // Complete Signal is False
      AN    #Cpu_Run_Pulse;
      JNB   _FWD;
      CALL SFC   20 (
           SRCBLK                   := #First_Stn,
           RET_VAL                  := #Ret,
           DSTBLK                   := #Mask);

NETWORK
TITLE =Clear Source Data Area


      CALL SFC   21 (
           IN0                      := #Fill_Source,// "Zero"
           RET_VAL                  := #Ret,
           OUT1                     := #First_Stn);// Transfer to First Station Area

NETWORK
TITLE =Fwd Block Move to Second Station Area


      CALL SFC   20 (
           SRCBLK                   := #Mask,
           RET_VAL                  := #Ret,
           DSTBLK                   := #Second_Stn);

NETWORK
TITLE =Clear Mask Data Area


      CALL SFC   21 (
           IN0                      := #Fill_Source,// "Zero"
           RET_VAL                  := #Ret,
           OUT1                     := #Mask);// Transfer to Mask Area
_FWD: NOP   0;
NETWORK
TITLE =Rev Block Move to Mask Area

      A     #RET_Pulse; // External Return Operation Signal
      AN    #Complete; // Complete Signal is False
      AN    #Cpu_Run_Pulse;
      JNB   _REV;
      CALL SFC   20 (
           SRCBLK                   := #Second_Stn,
           RET_VAL                  := #Ret,
           DSTBLK                   := #Mask);

NETWORK
TITLE =Clear Source Data Area


      CALL SFC   21 (
           IN0                      := #Fill_Source,// "Zero"
           RET_VAL                  := #Ret,
           OUT1                     := #Second_Stn);// Transfer to Second Station Area

NETWORK
TITLE =Rev Block Move to First Station Area


      CALL SFC   20 (
           SRCBLK                   := #Mask,
           RET_VAL                  := #Ret,
           DSTBLK                   := #First_Stn);

NETWORK
TITLE =Clear Mask Data Area


      CALL SFC   21 (
           IN0                      := #Fill_Source,// "Zero"
           RET_VAL                  := #Ret,
           OUT1                     := #Mask);// Transfer to Mask Area
_REV: NOP   0;
NETWORK
TITLE =Set Complete Signal

      S     #Complete;
_End: NOP   0;
END_FUNCTION_BLOCK

FUNCTION_BLOCK FB 470
TITLE =HMI Body Type Modify Variables Program
AUTHOR : HMC
FAMILY : HMI
NAME : HMI
VERSION : 1.0


VAR_INPUT
  Station : INT ;
  HMI_Disp_DB : INT ;
  HMI_Disp_Add : INT ;
  CType_DB : INT ;
  CType_Start_Add : INT ;
  Byte_per_Stn : INT ;
  M_Modify_OK : BOOL ;
  SS_CCR_On : BOOL ;
  PB_Set : BOOL ;
  PB_Reset : BOOL ;
END_VAR
VAR_OUTPUT
  LP_CCR_On : BOOL ;
  LP_Modify_On : BOOL ;
END_VAR
VAR
  Source_Data : WORD ;
  Modify_Data : WORD ;
  Pre_Station : INT ;
  Station_PLS : BOOL ;
  Source_Add : INT ;
  SFC20_Ret : INT ;
  Fill_Source : WORD ;
END_VAR
VAR_TEMP
  Source_Area : ANY ;
  Modify_Area : ANY ;
END_VAR
BEGIN
NETWORK
TITLE =FAC On Lamp Program

      A     #SS_CCR_On;
      =     #LP_CCR_On;
NETWORK
TITLE =Operation Pulse

      L     #Station; // Station Select Data
      L     0; // Is Not Zero
      <>I   ;
      JNB   _End; // Jump to End
NETWORK
TITLE =Modify On Lamp Program
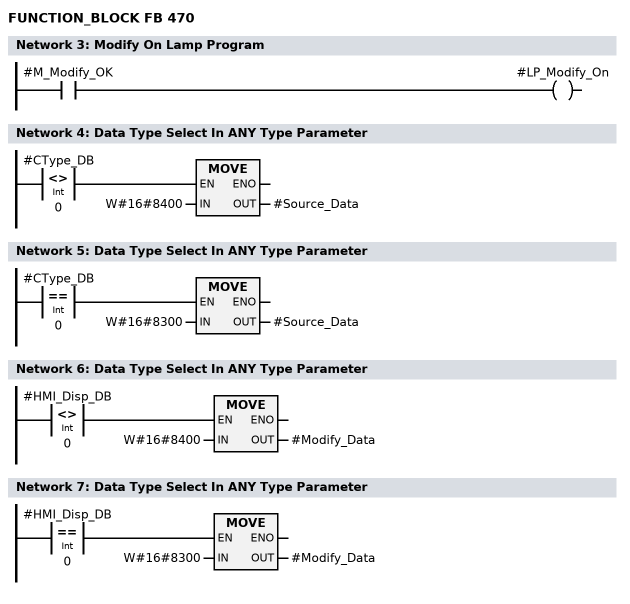

      A     #M_Modify_OK;
      =     #LP_Modify_On;
NETWORK
TITLE =Data Type Select In ANY Type Parameter

      A(    ; // If Source DB is Not Zero
      L     #CType_DB;
      L     0;
      <>I   ;
      )     ;
      JNB   _B01; // Jump to Next Step
      L     W#16#8400; // Load "8400" _ Means "DB Area"
      T     #Source_Data; // Transfer to Data_Type
_B01: NOP   0;
NETWORK
TITLE =Data Type Select In ANY Type Parameter

      A(    ; // If DB_NO is Zero
      L     #CType_DB;
      L     0;
      ==I   ;
      )     ;
      JNB   _B02; // Jump to Next Step
      L     W#16#8300; // Load "8300" _ Means "Bit Memory Area"
      T     #Source_Data; // Transfer to Data_Type
_B02: NOP   0;
NETWORK
TITLE =Data Type Select In ANY Type Parameter

      A(    ; // If Source DB is Not Zero
      L     #HMI_Disp_DB;
      L     0;
      <>I   ;
      )     ;
      JNB   _B03; // Jump to Next Step
      L     W#16#8400; // Load "8400" _ Means "DB Area"
      T     #Modify_Data; // Transfer to Data_Type
_B03: NOP   0;
NETWORK
TITLE =Data Type Select In ANY Type Parameter

      A(    ; // If DB_NO is Zero
      L     #HMI_Disp_DB;
      L     0;
      ==I   ;
      )     ;
      JNB   _B04; // Jump to Next Step
      L     W#16#8300; // Load "8300" _ Means "Bit Memory Area"
      T     #Modify_Data; // Transfer to Data_Type
_B04: NOP   0;
NETWORK
TITLE =Source Area Start Address Calculate Porgram

      L     #Station; // Station Amount - 1
      L     1;
      -I    ;
      L     #Byte_per_Stn; // Multi Length Per Station
      *I    ;
      L     #CType_Start_Add;
      +I    ;
      T     #Source_Add;
NETWORK
TITLE =Make a "ANY" Type Data

      LAR1  P##Source_Area; // Load 1st Station Address of ANY Pointer In "AR1"

      L     B#16#10; // Load Syntax ID For S7 "10"
      T     LB [AR1,P#0.0]; // Transfer ID to the ANY Pointer

      L     B#16#2; // Load Data Type _ "2" means "BYTE"
      T     LB [AR1,P#1.0]; // Transfer Data Type to the ANY Pointer

      L     #Byte_per_Stn; // Load the Length of Source Data
      T     LW [AR1,P#2.0]; // Transfer the Numbers to the ANY Pointer

      L     #CType_DB; // Load DB Number _ "0" means don't use "DB"
      T     LW [AR1,P#4.0]; // Transfer the Numbers to the ANY Pointer

      L     #Source_Data; // Load Data Type _ "83" means "Bit Memory" Area
      T     LW [AR1,P#6.0]; //                  "84" means "DB" Area

      L     #Source_Add; // Load Start Address
      SLW   3; // Shift Left Word _ "3" Bit
      T     LW [AR1,P#8.0]; // Transfer the Address to the ANY Pointer

      LAR1  P##Modify_Area; // Load 2nd Station Address of ANY Pointer In "AR1"

      L     B#16#10; //Load Syntax ID For S7 "10"
      T     LB [AR1,P#0.0]; //Load Syntax ID For S7 "10"

      L     B#16#2; //  Load Data Type _ "2" means "BYTE"
      T     LB [AR1,P#1.0]; // Transfer Data Type to the ANY Pointer

      L     #Byte_per_Stn; // Load the Length of Target Data
      T     LW [AR1,P#2.0]; // Transfer the Numbers to the ANY Pointer

      L     #HMI_Disp_DB; // Load DB Number _ "0" means don't use "DB"
      T     LW [AR1,P#4.0]; // Transfer the Numbers to the ANY Pointer

      L     #Modify_Data; // Load Data Type _ "83" means "Bit Memory" Area
      T     LW [AR1,P#6.0]; //                  "84" means "DB" Area

      L     #HMI_Disp_Add; //  Load Start Address
      SLW   3; // Shift Left Word _ "3" Bit
      T     LW [AR1,P#8.0]; // Transfer the Address to the ANY Pointer

NETWORK
TITLE =Copy To Modify Area Program

      L     #Station;
      L     #Pre_Station;
      <>I   ;
      JNB   _B05;
NETWORK
TITLE =Copy To Previous Station No Program

      L     #Station;
      T     #Pre_Station;
NETWORK
TITLE =Block Move to Modify Area


      CALL SFC   20 (
           SRCBLK                   := #Source_Area,
           RET_VAL                  := #SFC20_Ret,
           DSTBLK                   := #Modify_Area);
_B05: NOP   0;
NETWORK
TITLE =Data Clear Program

      A     #M_Modify_OK;
      A     #PB_Reset;
      JNB   _B06;
NETWORK
TITLE =Clear Source Data Area


      CALL SFC   21 (
           IN0                      := #Fill_Source,// "Zero"
           RET_VAL                  := #SFC20_Ret,
           OUT1                     := #Source_Area);// Transfer to First Station Area

NETWORK
TITLE =Clear Source Data Area


      CALL SFC   21 (
           IN0                      := #Fill_Source,// "Zero"
           RET_VAL                  := #SFC20_Ret,
           OUT1                     := #Modify_Area);// Transfer to First Station Area
_B06: NOP   0;
NETWORK
TITLE =Data Clear Program

      A     #M_Modify_OK;
      A     #PB_Set;
      JNB   _B07;
NETWORK
TITLE =Block Move to Modify Area


      CALL SFC   20 (
           SRCBLK                   := #Modify_Area,
           RET_VAL                  := #SFC20_Ret,
           DSTBLK                   := #Source_Area);
_B07: NOP   0;
NETWORK
TITLE =


_End: NOP   0;

END_FUNCTION_BLOCK

FUNCTION_BLOCK FB 475
TITLE =ProfiBus DP Communication Fault Variables Program
AUTHOR : HMC
FAMILY : Drive
NAME : Drive
VERSION : 1.0


VAR_INPUT
  M_Check_Active : BOOL ;
  DP_Not_Pre_Byte : BYTE ;	//Startadress Outputs from HW-Konfig
  DP_Error_Byte : BYTE ;	//Startadress Inputs from HW-Konfig
  M_Error_Rst : BOOL ;
END_VAR
VAR_OUTPUT
  Node0_Fault : BOOL ;
  Node1_Fault : BOOL ;
  Node2_Fault : BOOL ;
  Node3_Fault : BOOL ;
  Node4_Fault : BOOL ;
  Node5_Fault : BOOL ;
  Node6_Fault : BOOL ;
  Node7_Fault : BOOL ;
END_VAR
VAR
  Pre_Arr : ARRAY  [0 .. 7 ] OF BOOL ;
  Fault_Arr : ARRAY  [0 .. 7 ] OF BOOL ;
  node_0_err : SFB 4;
  node_1_err : SFB 4;
  node_2_err : SFB 4;
  node_3_err : SFB 4;
  node_4_err : SFB 4;
  node_5_err : SFB 4;
  node_6_err : SFB 4;
  node_7_err : SFB 4;
END_VAR
VAR_TEMP
  Ret : INT ;
END_VAR
BEGIN
NETWORK
TITLE =DP Fault Byte Move To DP Fault Array
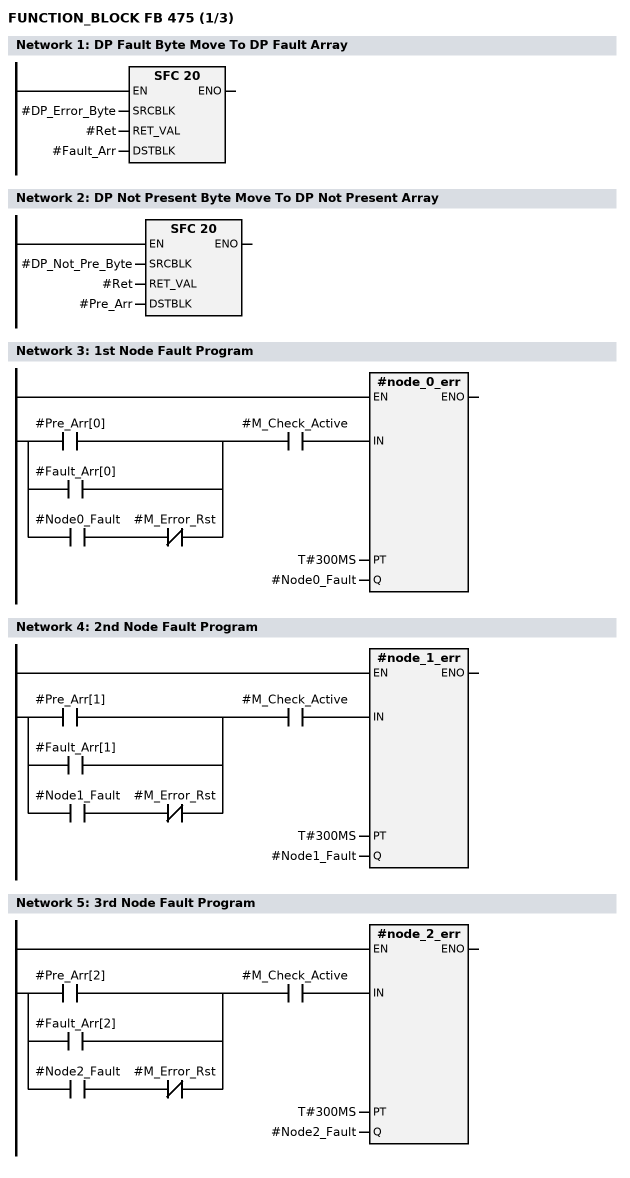

      CALL SFC   20 (
           SRCBLK                   := #DP_Error_Byte,
           RET_VAL                  := #Ret,
           DSTBLK                   := #Fault_Arr);
      NOP   0;
NETWORK
TITLE =DP Not Present Byte Move To DP Not Present Array

      CALL SFC   20 (
           SRCBLK                   := #DP_Not_Pre_Byte,
           RET_VAL                  := #Ret,
           DSTBLK                   := #Pre_Arr);
      NOP   0;
NETWORK
TITLE =1st Node Fault Program

      A(    ;
      O     #Pre_Arr[0];
      O     #Fault_Arr[0];
      O     ;
      A     #Node0_Fault;
      AN    #M_Error_Rst;
      )     ;
      A     #M_Check_Active;
      =     L      2.0;
      BLD   103;
      CALL #node_0_err (
           IN                       := L      2.0,
           PT                       := T#300MS,
           Q                        := #Node0_Fault);

      NOP   0;
NETWORK
TITLE =2nd Node Fault Program

      A(    ;
      O     #Pre_Arr[1];
      O     #Fault_Arr[1];
      O     ;
      A     #Node1_Fault;
      AN    #M_Error_Rst;
      )     ;
      A     #M_Check_Active;
      =     L      2.0;
      BLD   103;
      CALL #node_1_err (
           IN                       := L      2.0,
           PT                       := T#300MS,
           Q                        := #Node1_Fault);

      NOP   0;
NETWORK
TITLE =3rd Node Fault Program

      A(    ;
      O     #Pre_Arr[2];
      O     #Fault_Arr[2];
      O     ;
      A     #Node2_Fault;
      AN    #M_Error_Rst;
      )     ;
      A     #M_Check_Active;
      =     L      2.0;
      BLD   103;
      CALL #node_2_err (
           IN                       := L      2.0,
           PT                       := T#300MS,
           Q                        := #Node2_Fault);

      NOP   0;
NETWORK
TITLE =4th Node Fault Program
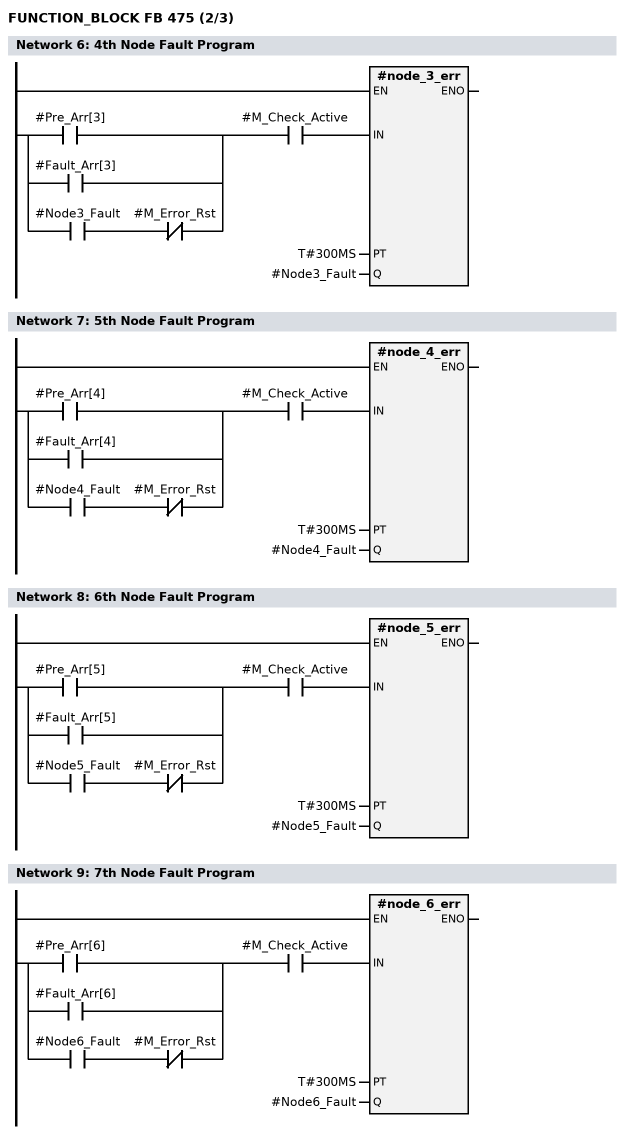

      A(    ;
      O     #Pre_Arr[3];
      O     #Fault_Arr[3];
      O     ;
      A     #Node3_Fault;
      AN    #M_Error_Rst;
      )     ;
      A     #M_Check_Active;
      =     L      2.0;
      BLD   103;
      CALL #node_3_err (
           IN                       := L      2.0,
           PT                       := T#300MS,
           Q                        := #Node3_Fault);

      NOP   0;
NETWORK
TITLE =5th Node Fault Program

      A(    ;
      O     #Pre_Arr[4];
      O     #Fault_Arr[4];
      O     ;
      A     #Node4_Fault;
      AN    #M_Error_Rst;
      )     ;
      A     #M_Check_Active;
      =     L      2.0;
      BLD   103;
      CALL #node_4_err (
           IN                       := L      2.0,
           PT                       := T#300MS,
           Q                        := #Node4_Fault);

      NOP   0;
NETWORK
TITLE =6th Node Fault Program

      A(    ;
      O     #Pre_Arr[5];
      O     #Fault_Arr[5];
      O     ;
      A     #Node5_Fault;
      AN    #M_Error_Rst;
      )     ;
      A     #M_Check_Active;
      =     L      2.0;
      BLD   103;
      CALL #node_5_err (
           IN                       := L      2.0,
           PT                       := T#300MS,
           Q                        := #Node5_Fault);

      NOP   0;
NETWORK
TITLE =7th Node Fault Program

      A(    ;
      O     #Pre_Arr[6];
      O     #Fault_Arr[6];
      O     ;
      A     #Node6_Fault;
      AN    #M_Error_Rst;
      )     ;
      A     #M_Check_Active;
      =     L      2.0;
      BLD   103;
      CALL #node_6_err (
           IN                       := L      2.0,
           PT                       := T#300MS,
           Q                        := #Node6_Fault);

      NOP   0;
NETWORK
TITLE =8th Node Fault Program
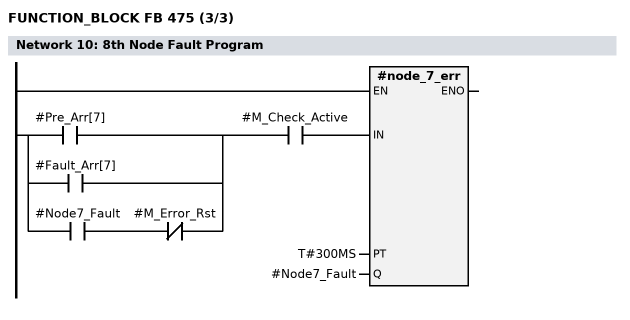

      A(    ;
      O     #Pre_Arr[7];
      O     #Fault_Arr[7];
      O     ;
      A     #Node7_Fault;
      AN    #M_Error_Rst;
      )     ;
      A     #M_Check_Active;
      =     L      2.0;
      BLD   103;
      CALL #node_7_err (
           IN                       := L      2.0,
           PT                       := T#300MS,
           Q                        := #Node7_Fault);

      NOP   0;
END_FUNCTION_BLOCK

FUNCTION_BLOCK FB 512
TITLE =Car Type Variables Program
AUTHOR : HMC
FAMILY : Car_Type
NAME : Car_Type
VERSION : 1.0


VAR_INPUT
  Stn_Vin_No : DINT ;	//Startadress Inputs from HW-Konfig
  Stn_Bt_1Word : WORD ;
  Stn_Bt_2Word : WORD ;
  Stn_Bt_3Word : WORD ;
  Stn_Bt_4Word : WORD ;
  Stn_Bt_5Word_Sp : WORD ;
  Stn_Bt_6Word_Sp : WORD ;
END_VAR
VAR_OUTPUT
  M_BType_On : BOOL ;
  M_BType_None : BOOL ;
  M_Bypass_BType : BOOL ;
  M_BType_TL : BOOL ;
  M_BType_LM : BOOL ;
  M_BType_SP1 : BOOL ;
  M_BType_SP2 : BOOL ;
  M_BType_SP3 : BOOL ;
  M_BType_DOM : BOOL ;
  M_BType_EXP : BOOL ;
  Robot_Prog_No : INT ;
END_VAR
VAR
  STN_Btype_1Arr : ARRAY  [0 .. 15 ] OF BOOL ;
  STN_Btype_2Arr : ARRAY  [0 .. 15 ] OF BOOL ;
  STN_Btype_3Arr : ARRAY  [0 .. 15 ] OF BOOL ;
  STN_Btype_4Arr : ARRAY  [0 .. 15 ] OF BOOL ;
  STN_Btype_5Arr : ARRAY  [0 .. 15 ] OF BOOL ;
  STN_Btype_6Arr : ARRAY  [0 .. 15 ] OF BOOL ;
  STN_1st_BT_On : BOOL ;
  STN_2nd_BT_On : BOOL ;
  STN_3rd_BT_On : BOOL ;
  STN_4th_BT_On : BOOL ;
  STN_5th_BT_On : BOOL ;
  STN_6th_BT_On : BOOL ;
  STN_7th_BT_On : BOOL ;
  STN_8th_BT_On : BOOL ;
  STN_9th_BT_On : BOOL ;
  STN_10th_BT_On : BOOL ;
  STN_11th_BT_On : BOOL ;
  STN_12th_BT_On : BOOL ;
  STN_1st_BT_Off : BOOL ;
  BLKMove_Ret : INT ;
  VIN_1BCD : WORD ;
  VIN_2BCD : WORD ;
  VIN_1Int : INT ;
  VIN_2Int : INT ;
END_VAR
BEGIN
NETWORK
TITLE =Station Body Type Data Change to 16-bit array

      CALL SFC   20 (
           SRCBLK                   := #Stn_Bt_1Word,
           RET_VAL                  := #BLKMove_Ret,
           DSTBLK                   := #STN_Btype_1Arr);
      NOP   0;
NETWORK
TITLE =Station Body Type Data Change to 16-bit array

      CALL SFC   20 (
           SRCBLK                   := #Stn_Bt_2Word,
           RET_VAL                  := #BLKMove_Ret,
           DSTBLK                   := #STN_Btype_2Arr);
      NOP   0;
NETWORK
TITLE =Station Body Type Data Change to 16-bit array

      CALL SFC   20 (
           SRCBLK                   := #Stn_Bt_3Word,
           RET_VAL                  := #BLKMove_Ret,
           DSTBLK                   := #STN_Btype_3Arr);
      NOP   0;
NETWORK
TITLE =Station Body Type Data Change to 16-bit array

      CALL SFC   20 (
           SRCBLK                   := #Stn_Bt_4Word,
           RET_VAL                  := #BLKMove_Ret,
           DSTBLK                   := #STN_Btype_4Arr);
      NOP   0;
NETWORK
TITLE =Station Body Type Data Change to 16-bit array

      CALL SFC   20 (
           SRCBLK                   := #Stn_Bt_5Word_Sp,
           RET_VAL                  := #BLKMove_Ret,
           DSTBLK                   := #STN_Btype_5Arr);
      NOP   0;
NETWORK
TITLE =Station Body Type Data Change to 16-bit array

      CALL SFC   20 (
           SRCBLK                   := #Stn_Bt_6Word_Sp,
           RET_VAL                  := #BLKMove_Ret,
           DSTBLK                   := #STN_Btype_6Arr);
      NOP   0;
NETWORK
TITLE =공정 1차종

      AN    OV;
      A(    ;
      O     #STN_Btype_1Arr[0];
      O     #STN_Btype_1Arr[1];
      O     #STN_Btype_1Arr[2];
      O     #STN_Btype_1Arr[3];
      O     #STN_Btype_1Arr[4];
      )     ;
      =     #STN_1st_BT_On;
NETWORK
TITLE =공정 2차종

      AN    OV;
      A(    ;
      O     #STN_Btype_1Arr[5];
      O     #STN_Btype_1Arr[6];
      O     #STN_Btype_1Arr[7];
      O     #STN_Btype_1Arr[8];
      )     ;
      =     #STN_2nd_BT_On;
NETWORK
TITLE =공정 3차종

      AN    OV;
      A(    ;
      O     #STN_Btype_1Arr[9];
      O     #STN_Btype_1Arr[10];
      )     ;
      =     #STN_3rd_BT_On;
NETWORK
TITLE =공정 4차종

      AN    OV;
      A(    ;
      O     #STN_Btype_1Arr[11];
      O     #STN_Btype_1Arr[12];
      O     #STN_Btype_1Arr[13];
      O     #STN_Btype_1Arr[14];
      O     #STN_Btype_1Arr[15];
      O     #STN_Btype_2Arr[0];
      O     #STN_Btype_2Arr[1];
      O     #STN_Btype_2Arr[2];
      O     #STN_Btype_2Arr[3];
      O     #STN_Btype_2Arr[4];
      O     #STN_Btype_2Arr[5];
      )     ;
      =     #STN_4th_BT_On;
NETWORK
TITLE =공정 5차종

      AN    OV;
      A(    ;
      O     #STN_Btype_2Arr[6];
      O     #STN_Btype_2Arr[7];
      )     ;
      =     #STN_5th_BT_On;
NETWORK
TITLE =공정 6차종

      AN    OV;
      A(    ;
      O     #STN_Btype_2Arr[8];
      O     #STN_Btype_2Arr[9];
      O     #STN_Btype_2Arr[10];
      O     #STN_Btype_2Arr[11];
      O     #STN_Btype_2Arr[12];
      O     #STN_Btype_2Arr[13];
      O     #STN_Btype_2Arr[14];
      O     #STN_Btype_2Arr[15];
      )     ;
      =     #STN_6th_BT_On;
NETWORK
TITLE =공정 7차종

      AN    OV;
      A(    ;
      O     #STN_Btype_3Arr[0];
      O     #STN_Btype_3Arr[1];
      )     ;
      =     #STN_7th_BT_On;
NETWORK
TITLE =공정 8차종

      AN    OV;
      A(    ;
      O     #STN_Btype_3Arr[2];
      O     #STN_Btype_3Arr[3];
      O     #STN_Btype_3Arr[6];
      )     ;
      =     #STN_8th_BT_On;
NETWORK
TITLE =공정 9차종

      AN    OV;
      A(    ;
      O     #STN_Btype_3Arr[4];
      O     #STN_Btype_3Arr[5];
      )     ;
      =     #STN_9th_BT_On;
NETWORK
TITLE =공정 10차종

      AN    OV;
      A(    ;
      O     #STN_Btype_3Arr[6];
      O     #STN_Btype_3Arr[7];
      ON    #STN_10th_BT_On;
      )     ;
      =     #STN_10th_BT_On;
NETWORK
TITLE =공정 11차종

      AN    OV;
      A(    ;
      O     #STN_Btype_3Arr[8];
      O     #STN_Btype_3Arr[9];
      O     #STN_Btype_3Arr[10];
      O     #STN_Btype_3Arr[11];
      O     #STN_Btype_3Arr[12];
      O     #STN_Btype_3Arr[13];
      O     #STN_Btype_3Arr[14];
      O     #STN_Btype_3Arr[15];
      O     #STN_Btype_4Arr[0];
      O     #STN_Btype_4Arr[1];
      O     #STN_Btype_4Arr[2];
      O     #STN_Btype_4Arr[3];
      O     #STN_Btype_4Arr[4];
      O     #STN_Btype_4Arr[5];
      O     #STN_Btype_4Arr[6];
      O     #STN_Btype_4Arr[7];
      O     #STN_Btype_4Arr[8];
      O     #STN_Btype_4Arr[9];
      )     ;
      =     #STN_11th_BT_On;
NETWORK
TITLE =공정 차종 있음
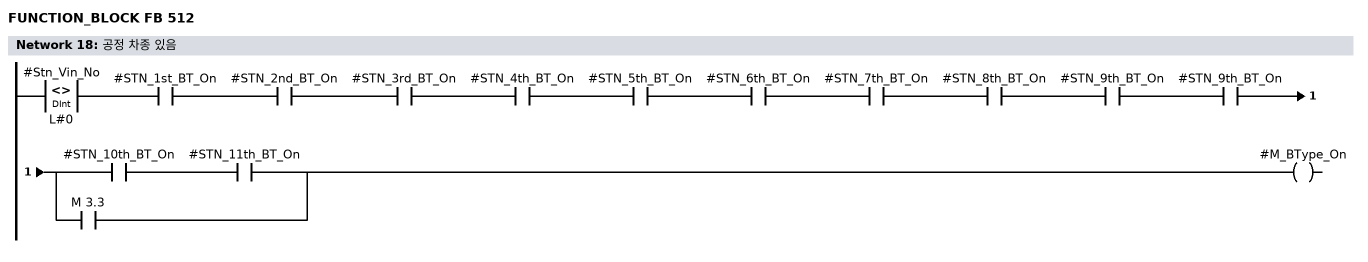

      A(    ;
      L     #Stn_Vin_No;
      L     L#0;
      <>D   ;
      )     ;
      A     #STN_1st_BT_On;
      A     #STN_2nd_BT_On;
      A     #STN_3rd_BT_On;
      A     #STN_4th_BT_On;
      A     #STN_5th_BT_On;
      A     #STN_6th_BT_On;
      A     #STN_7th_BT_On;
      A     #STN_8th_BT_On;
      A     #STN_9th_BT_On;
      A     #STN_9th_BT_On;
      A(    ;
      A     #STN_10th_BT_On;
      A     #STN_11th_BT_On;
      O     M      3.3;
      )     ;
      =     #M_BType_On;
NETWORK
TITLE =1차종 없음

      AN    OV;
      AN    #STN_Btype_1Arr[0];
      AN    #STN_Btype_1Arr[1];
      AN    #STN_Btype_1Arr[2];
      AN    #STN_Btype_1Arr[3];
      AN    #STN_Btype_1Arr[4];
      =     #STN_1st_BT_Off;
NETWORK
TITLE =공정 차종 없음
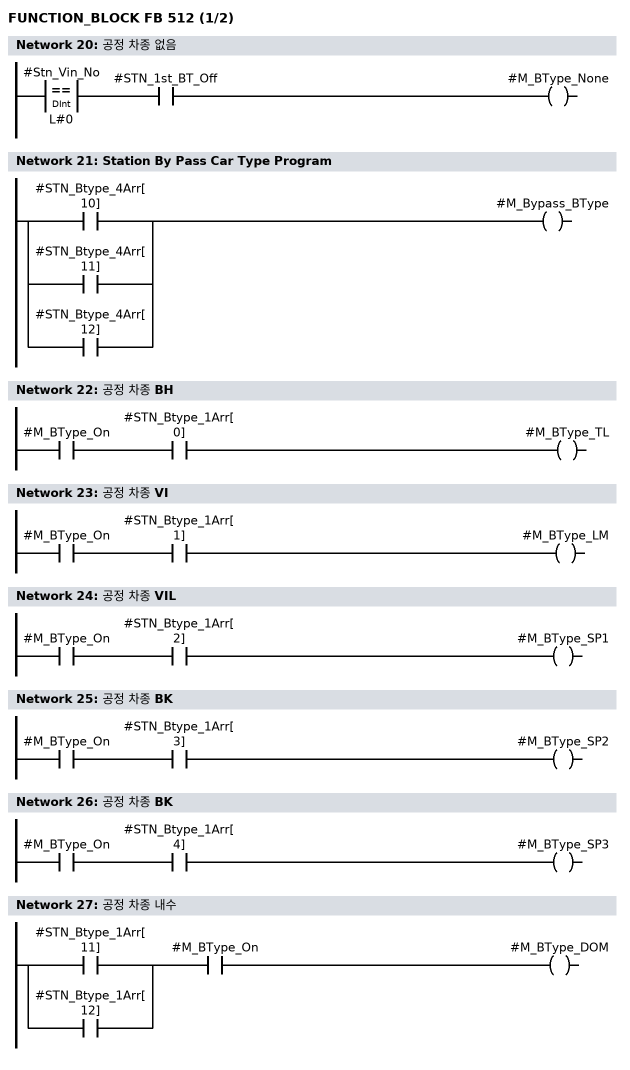

      A(    ;
      L     #Stn_Vin_No;
      L     L#0;
      ==D   ;
      )     ;
      A     #STN_1st_BT_Off;
      =     #M_BType_None;
NETWORK
TITLE =Station By Pass Car Type Program

      O     #STN_Btype_4Arr[10];
      O     #STN_Btype_4Arr[11];
      O     #STN_Btype_4Arr[12];
      =     #M_Bypass_BType;
NETWORK
TITLE =공정 차종 BH

      A     #M_BType_On;
      A     #STN_Btype_1Arr[0];
      =     #M_BType_TL;
NETWORK
TITLE =공정 차종 VI

      A     #M_BType_On;
      A     #STN_Btype_1Arr[1];
      =     #M_BType_LM;
NETWORK
TITLE =공정 차종 VIL

      A     #M_BType_On;
      A     #STN_Btype_1Arr[2];
      =     #M_BType_SP1;
NETWORK
TITLE =공정 차종 BK

      A     #M_BType_On;
      A     #STN_Btype_1Arr[3];
      =     #M_BType_SP2;
NETWORK
TITLE =공정 차종 BK

      A     #M_BType_On;
      A     #STN_Btype_1Arr[4];
      =     #M_BType_SP3;
NETWORK
TITLE =공정 차종 내수

      A(    ;
      O     #STN_Btype_1Arr[11];
      O     #STN_Btype_1Arr[12];
      )     ;
      A     #M_BType_On;
      =     #M_BType_DOM;
NETWORK
TITLE =공정 차종 수출
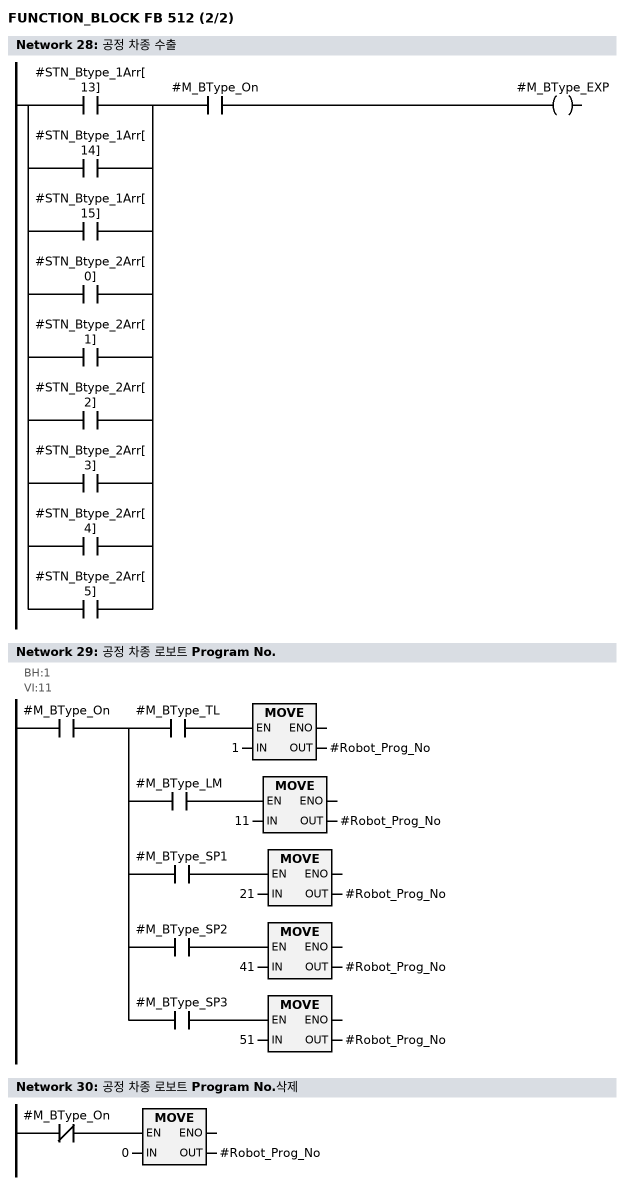

      A(    ;
      O     #STN_Btype_1Arr[13];
      O     #STN_Btype_1Arr[14];
      O     #STN_Btype_1Arr[15];
      O     #STN_Btype_2Arr[0];
      O     #STN_Btype_2Arr[1];
      O     #STN_Btype_2Arr[2];
      O     #STN_Btype_2Arr[3];
      O     #STN_Btype_2Arr[4];
      O     #STN_Btype_2Arr[5];
      )     ;
      A     #M_BType_On;
      =     #M_BType_EXP;
NETWORK
TITLE =공정 차종 로보트 Program No.
//BH:1
//VI:11
      A     #M_BType_On;
      =     L      0.0;
      A     L      0.0;
      A     #M_BType_TL;
      JNB   _001;
      L     1;
      T     #Robot_Prog_No;
_001: NOP   0;
      A     L      0.0;
      A     #M_BType_LM;
      JNB   _002;
      L     11;
      T     #Robot_Prog_No;
_002: NOP   0;
      A     L      0.0;
      A     #M_BType_SP1;
      JNB   _003;
      L     21;
      T     #Robot_Prog_No;
_003: NOP   0;
      A     L      0.0;
      A     #M_BType_SP2;
      JNB   _004;
      L     41;
      T     #Robot_Prog_No;
_004: NOP   0;
      A     L      0.0;
      A     #M_BType_SP3;
      JNB   _005;
      L     51;
      T     #Robot_Prog_No;
_005: NOP   0;
NETWORK
TITLE =공정 차종 로보트 Program No.삭제

      AN    #M_BType_On;
      JNB   _006;
      L     0;
      T     #Robot_Prog_No;
_006: NOP   0;
END_FUNCTION_BLOCK

DATA_BLOCK DB 71
TITLE =
AUTHOR : SIMATIC
FAMILY : CPU_300
VERSION : 0.0

 FB 12
BEGIN
   REQ := FALSE;
   R := FALSE;
   ID := W#16#4;
   R_ID := DW#16#4;
   DONE := FALSE;
   ERROR := FALSE;
   STATUS := W#16#0;
   SD_1 := P#DB22.DBX 0.0 BYTE 180;
   LEN := W#16#B4;
   FB_ZUSTAND := B#16#0;
   REQ_SAVE := FALSE;
   R_SAVE := FALSE;
   ID_SAVE := W#16#0;
   R_ID_SAVE := DW#16#0;
   LEN_SAVE := W#16#0;
   SD_1_SAVE0 := W#16#0;
   SD_1_SAVE2 := W#16#0;
   SD_1_SAVE4 := W#16#0;
   SD_1_SAVE6 := W#16#0;
   SD_1_SAVE8 := W#16#0;
   HS_REQ_BYTE.rii := FALSE;
   HS_REQ_BYTE.nva := FALSE;
   HS_REQ_BYTE.ofs := FALSE;
   HS_REQ_BYTE.dir := FALSE;
   HS_REQ_BYTE.res := FALSE;
   HS_REQ_BYTE.roc := FALSE;
   HS_REQ_BYTE.nls := FALSE;
   HS_REQ_BYTE.rlo := FALSE;
   HS_RESP_BYTE.aii := FALSE;
   HS_RESP_BYTE.sns := FALSE;
   HS_RESP_BYTE.sqc := FALSE;
   HS_RESP_BYTE.ads := FALSE;
   HS_RESP_BYTE.aoc := FALSE;
   HS_RESP_BYTE.rs1 := FALSE;
   HS_RESP_BYTE.cnr := FALSE;
   HS_RESP_BYTE.rs2 := FALSE;
   HS_RESP_DSNR := B#16#0;
   HS_RESP_OFFSET := W#16#0;
   SD_1_WORD0 := W#16#0;
   SD_1_COUNT := W#16#0;
   SD_1_DBNUMMER := W#16#0;
   SD_1_DWORD6 := DW#16#0;
   SD_1_TYP := B#16#0;
   SFC_PARAM.LEN := W#16#0;
   SFC_PARAM.DB_NUMMER := W#16#0;
   SFC_PARAM.START := DW#16#0;
   BUFFER[0] := W#16#0;
   BUFFER[1] := W#16#0;
   BUFFER[2] := W#16#0;
   BUFFER[3] := W#16#0;
   BUFFER[4] := W#16#0;
   BUFFER[5] := W#16#0;
   BUFFER[6] := W#16#0;
   BUFFER[7] := W#16#0;
   BUFFER[8] := W#16#0;
   BUFFER[9] := W#16#0;
   BUFFER[10] := W#16#0;
   BUFFER[11] := W#16#0;
   BUFFER[12] := W#16#0;
   BUFFER[13] := W#16#0;
   BUFFER[14] := W#16#0;
   BUFFER[15] := W#16#0;
   BUFFER[16] := W#16#0;
   BUFFER[17] := W#16#0;
   BUFFER[18] := W#16#0;
   BUFFER[19] := W#16#0;
   BUFFER[20] := W#16#0;
   BUFFER[21] := W#16#0;
   BUFFER[22] := W#16#0;
   BUFFER[23] := W#16#0;
   BUFFER[24] := W#16#0;
   BUFFER[25] := W#16#0;
   BUFFER[26] := W#16#0;
   BUFFER[27] := W#16#0;
   BUFFER[28] := W#16#0;
   BUFFER[29] := W#16#0;
   BUFFER[30] := W#16#0;
   BUFFER[31] := W#16#0;
   BUFFER[32] := W#16#0;
   BUFFER[33] := W#16#0;
   BUFFER[34] := W#16#0;
   BUFFER[35] := W#16#0;
   BUFFER[36] := W#16#0;
   BUFFER[37] := W#16#0;
   BUFFER[38] := W#16#0;
   BUFFER[39] := W#16#0;
   BUFFER[40] := W#16#0;
   BUFFER[41] := W#16#0;
   BUFFER[42] := W#16#0;
   BUFFER[43] := W#16#0;
   BUFFER[44] := W#16#0;
   BUFFER[45] := W#16#0;
   BUFFER[46] := W#16#0;
   BUFFER[47] := W#16#0;
   BUFFER[48] := W#16#0;
   BUFFER[49] := W#16#0;
   BUFFER[50] := W#16#0;
   BUFFER[51] := W#16#0;
   BUFFER[52] := W#16#0;
   BUFFER[53] := W#16#0;
   BUFFER[54] := W#16#0;
   BUFFER[55] := W#16#0;
   BUFFER[56] := W#16#0;
   BUFFER[57] := W#16#0;
   BUFFER[58] := W#16#0;
   BUFFER[59] := W#16#0;
   BUFFER[60] := W#16#0;
   BUFFER[61] := W#16#0;
   BUFFER[62] := W#16#0;
   BUFFER[63] := W#16#0;
   BUFFER[64] := W#16#0;
   BUFFER[65] := W#16#0;
   BUFFER[66] := W#16#0;
   BUFFER[67] := W#16#0;
   BUFFER[68] := W#16#0;
   BUFFER[69] := W#16#0;
   BUFFER[70] := W#16#0;
   BUFFER[71] := W#16#0;
   BUFFER[72] := W#16#0;
   BUFFER[73] := W#16#0;
   BUFFER[74] := W#16#0;
   BUFFER[75] := W#16#0;
   BUFFER[76] := W#16#0;
   BUFFER[77] := W#16#0;
   BUFFER[78] := W#16#0;
   BUFFER[79] := W#16#0;
   BUFFER[80] := W#16#0;
   BUFFER[81] := W#16#0;
   BUFFER[82] := W#16#0;
   BUFFER[83] := W#16#0;
   BUFFER[84] := W#16#0;
   BUFFER[85] := W#16#0;
   BUFFER[86] := W#16#0;
   BUFFER[87] := W#16#0;
   BUFFER[88] := W#16#0;
   BUFFER[89] := W#16#0;
   BUFFER[90] := W#16#0;
   BUFFER[91] := W#16#0;
   BUFFER[92] := W#16#0;
   BUFFER[93] := W#16#0;
   BUFFER[94] := W#16#0;
   BUFFER[95] := W#16#0;
   BUFFER[96] := W#16#0;
   BUFFER[97] := W#16#0;
   BUFFER[98] := W#16#0;
   BUFFER[99] := W#16#0;
   BUFFER[100] := W#16#0;
   BUFFER[101] := W#16#0;
   BUFFER[102] := W#16#0;
   BUFFER[103] := W#16#0;
   BUFFER[104] := W#16#0;
   BUFFER[105] := W#16#0;
   BUFFER[106] := W#16#0;
   BUFFER[107] := W#16#0;
   BUFFER[108] := W#16#0;
   BUFFER[109] := W#16#0;
   BUFFER[110] := W#16#0;
   BUFFER[111] := W#16#0;
   BUFFER[112] := W#16#0;
   BUFFER[113] := W#16#0;
   BUFFER[114] := W#16#0;
   BUFFER[115] := W#16#0;
   BUFFER[116] := W#16#0;
   BUFFER[117] := W#16#0;
   BUFFER[118] := W#16#0;
   BUFFER[119] := W#16#0;
   REASON_FOR_CLOSE := B#16#0;
   DS_NR := B#16#0;
   PARAM_OFFSET := B#16#0;
   MAX_PUFF_LEN_SAVE := W#16#0;
   TYP_BOOL := FALSE;
   KANAL_PROBLEM := FALSE;
   KOMM_PROBLEM := FALSE;
   SEND_STARTED := FALSE;
   RECV_STARTED := FALSE;
   RESET_REQUEST := FALSE;
   RESET_EXECUTED := FALSE;
   DS200_BUSY := FALSE;
   MAX_DATA_LEN := W#16#0;
   LADDR_PTR := DW#16#0;
   FC_DATA_LEN := W#16#0;
   LADDR := W#16#0;
   SLEEP := B#16#0;
   SLEEP_EXT := B#16#0;
   ID_CLOSE := W#16#0;
   FB_KENNUNG := B#16#F1;
   RESERVE := B#16#0;
   ZUSTAND_WEICHE := B#16#2;
   SFB_AUFRUF.REQ := TRUE;
   SFB_AUFRUF.R := FALSE;
   SFB_AUFRUF.ID := W#16#4;
   SFB_AUFRUF.R_ID := DW#16#4;
   SFB_AUFRUF.DONE := FALSE;
   SFB_AUFRUF.ERROR := FALSE;
   SFB_AUFRUF.STATUS := W#16#19;
   SFB_AUFRUF.SD_1 := P#DB22.DBX 0.0 BYTE 180;
   SFB_AUFRUF.LEN := W#16#B4;
   SFB_AUFRUF.INDEX := W#16#101;
   ZUSTAND_WEICHE_1 := B#16#CA;
END_DATA_BLOCK

DATA_BLOCK DB 72
TITLE =
AUTHOR : SIMATIC
FAMILY : CPU_300
VERSION : 0.0

 FB 12
BEGIN
   REQ := FALSE;
   R := FALSE;
   ID := W#16#12;
   R_ID := DW#16#12;
   DONE := FALSE;
   ERROR := FALSE;
   STATUS := W#16#0;
   SD_1 := P#DB16.DBX 0.0 BYTE 20;
   LEN := W#16#14;
   FB_ZUSTAND := B#16#0;
   REQ_SAVE := FALSE;
   R_SAVE := FALSE;
   ID_SAVE := W#16#0;
   R_ID_SAVE := DW#16#0;
   LEN_SAVE := W#16#0;
   SD_1_SAVE0 := W#16#0;
   SD_1_SAVE2 := W#16#0;
   SD_1_SAVE4 := W#16#0;
   SD_1_SAVE6 := W#16#0;
   SD_1_SAVE8 := W#16#0;
   HS_REQ_BYTE.rii := FALSE;
   HS_REQ_BYTE.nva := FALSE;
   HS_REQ_BYTE.ofs := FALSE;
   HS_REQ_BYTE.dir := FALSE;
   HS_REQ_BYTE.res := FALSE;
   HS_REQ_BYTE.roc := FALSE;
   HS_REQ_BYTE.nls := FALSE;
   HS_REQ_BYTE.rlo := FALSE;
   HS_RESP_BYTE.aii := FALSE;
   HS_RESP_BYTE.sns := FALSE;
   HS_RESP_BYTE.sqc := FALSE;
   HS_RESP_BYTE.ads := FALSE;
   HS_RESP_BYTE.aoc := FALSE;
   HS_RESP_BYTE.rs1 := FALSE;
   HS_RESP_BYTE.cnr := FALSE;
   HS_RESP_BYTE.rs2 := FALSE;
   HS_RESP_DSNR := B#16#0;
   HS_RESP_OFFSET := W#16#0;
   SD_1_WORD0 := W#16#0;
   SD_1_COUNT := W#16#0;
   SD_1_DBNUMMER := W#16#0;
   SD_1_DWORD6 := DW#16#0;
   SD_1_TYP := B#16#0;
   SFC_PARAM.LEN := W#16#0;
   SFC_PARAM.DB_NUMMER := W#16#0;
   SFC_PARAM.START := DW#16#0;
   BUFFER[0] := W#16#0;
   BUFFER[1] := W#16#0;
   BUFFER[2] := W#16#0;
   BUFFER[3] := W#16#0;
   BUFFER[4] := W#16#0;
   BUFFER[5] := W#16#0;
   BUFFER[6] := W#16#0;
   BUFFER[7] := W#16#0;
   BUFFER[8] := W#16#0;
   BUFFER[9] := W#16#0;
   BUFFER[10] := W#16#0;
   BUFFER[11] := W#16#0;
   BUFFER[12] := W#16#0;
   BUFFER[13] := W#16#0;
   BUFFER[14] := W#16#0;
   BUFFER[15] := W#16#0;
   BUFFER[16] := W#16#0;
   BUFFER[17] := W#16#0;
   BUFFER[18] := W#16#0;
   BUFFER[19] := W#16#0;
   BUFFER[20] := W#16#0;
   BUFFER[21] := W#16#0;
   BUFFER[22] := W#16#0;
   BUFFER[23] := W#16#0;
   BUFFER[24] := W#16#0;
   BUFFER[25] := W#16#0;
   BUFFER[26] := W#16#0;
   BUFFER[27] := W#16#0;
   BUFFER[28] := W#16#0;
   BUFFER[29] := W#16#0;
   BUFFER[30] := W#16#0;
   BUFFER[31] := W#16#0;
   BUFFER[32] := W#16#0;
   BUFFER[33] := W#16#0;
   BUFFER[34] := W#16#0;
   BUFFER[35] := W#16#0;
   BUFFER[36] := W#16#0;
   BUFFER[37] := W#16#0;
   BUFFER[38] := W#16#0;
   BUFFER[39] := W#16#0;
   BUFFER[40] := W#16#0;
   BUFFER[41] := W#16#0;
   BUFFER[42] := W#16#0;
   BUFFER[43] := W#16#0;
   BUFFER[44] := W#16#0;
   BUFFER[45] := W#16#0;
   BUFFER[46] := W#16#0;
   BUFFER[47] := W#16#0;
   BUFFER[48] := W#16#0;
   BUFFER[49] := W#16#0;
   BUFFER[50] := W#16#0;
   BUFFER[51] := W#16#0;
   BUFFER[52] := W#16#0;
   BUFFER[53] := W#16#0;
   BUFFER[54] := W#16#0;
   BUFFER[55] := W#16#0;
   BUFFER[56] := W#16#0;
   BUFFER[57] := W#16#0;
   BUFFER[58] := W#16#0;
   BUFFER[59] := W#16#0;
   BUFFER[60] := W#16#0;
   BUFFER[61] := W#16#0;
   BUFFER[62] := W#16#0;
   BUFFER[63] := W#16#0;
   BUFFER[64] := W#16#0;
   BUFFER[65] := W#16#0;
   BUFFER[66] := W#16#0;
   BUFFER[67] := W#16#0;
   BUFFER[68] := W#16#0;
   BUFFER[69] := W#16#0;
   BUFFER[70] := W#16#0;
   BUFFER[71] := W#16#0;
   BUFFER[72] := W#16#0;
   BUFFER[73] := W#16#0;
   BUFFER[74] := W#16#0;
   BUFFER[75] := W#16#0;
   BUFFER[76] := W#16#0;
   BUFFER[77] := W#16#0;
   BUFFER[78] := W#16#0;
   BUFFER[79] := W#16#0;
   BUFFER[80] := W#16#0;
   BUFFER[81] := W#16#0;
   BUFFER[82] := W#16#0;
   BUFFER[83] := W#16#0;
   BUFFER[84] := W#16#0;
   BUFFER[85] := W#16#0;
   BUFFER[86] := W#16#0;
   BUFFER[87] := W#16#0;
   BUFFER[88] := W#16#0;
   BUFFER[89] := W#16#0;
   BUFFER[90] := W#16#0;
   BUFFER[91] := W#16#0;
   BUFFER[92] := W#16#0;
   BUFFER[93] := W#16#0;
   BUFFER[94] := W#16#0;
   BUFFER[95] := W#16#0;
   BUFFER[96] := W#16#0;
   BUFFER[97] := W#16#0;
   BUFFER[98] := W#16#0;
   BUFFER[99] := W#16#0;
   BUFFER[100] := W#16#0;
   BUFFER[101] := W#16#0;
   BUFFER[102] := W#16#0;
   BUFFER[103] := W#16#0;
   BUFFER[104] := W#16#0;
   BUFFER[105] := W#16#0;
   BUFFER[106] := W#16#0;
   BUFFER[107] := W#16#0;
   BUFFER[108] := W#16#0;
   BUFFER[109] := W#16#0;
   BUFFER[110] := W#16#0;
   BUFFER[111] := W#16#0;
   BUFFER[112] := W#16#0;
   BUFFER[113] := W#16#0;
   BUFFER[114] := W#16#0;
   BUFFER[115] := W#16#0;
   BUFFER[116] := W#16#0;
   BUFFER[117] := W#16#0;
   BUFFER[118] := W#16#0;
   BUFFER[119] := W#16#0;
   REASON_FOR_CLOSE := B#16#0;
   DS_NR := B#16#0;
   PARAM_OFFSET := B#16#0;
   MAX_PUFF_LEN_SAVE := W#16#0;
   TYP_BOOL := FALSE;
   KANAL_PROBLEM := FALSE;
   KOMM_PROBLEM := FALSE;
   SEND_STARTED := FALSE;
   RECV_STARTED := FALSE;
   RESET_REQUEST := FALSE;
   RESET_EXECUTED := FALSE;
   DS200_BUSY := FALSE;
   MAX_DATA_LEN := W#16#0;
   LADDR_PTR := DW#16#0;
   FC_DATA_LEN := W#16#0;
   LADDR := W#16#0;
   SLEEP := B#16#0;
   SLEEP_EXT := B#16#0;
   ID_CLOSE := W#16#0;
   FB_KENNUNG := B#16#F1;
   RESERVE := B#16#0;
   ZUSTAND_WEICHE := B#16#2;
   SFB_AUFRUF.REQ := FALSE;
   SFB_AUFRUF.R := FALSE;
   SFB_AUFRUF.ID := W#16#12;
   SFB_AUFRUF.R_ID := DW#16#12;
   SFB_AUFRUF.DONE := FALSE;
   SFB_AUFRUF.ERROR := FALSE;
   SFB_AUFRUF.STATUS := W#16#0;
   SFB_AUFRUF.SD_1 := P#DB16.DBX 0.0 BYTE 20;
   SFB_AUFRUF.LEN := W#16#14;
   SFB_AUFRUF.INDEX := W#16#301;
   ZUSTAND_WEICHE_1 := B#16#CA;
END_DATA_BLOCK

DATA_BLOCK DB 73
TITLE =
AUTHOR : SIMATIC
FAMILY : CPU_300
VERSION : 0.0

 FB 12
BEGIN
   REQ := FALSE;
   R := FALSE;
   ID := W#16#14;
   R_ID := DW#16#14;
   DONE := FALSE;
   ERROR := FALSE;
   STATUS := W#16#0;
   SD_1 := P#DB17.DBX 0.0 BYTE 80;
   LEN := W#16#50;
   FB_ZUSTAND := B#16#0;
   REQ_SAVE := FALSE;
   R_SAVE := FALSE;
   ID_SAVE := W#16#0;
   R_ID_SAVE := DW#16#0;
   LEN_SAVE := W#16#0;
   SD_1_SAVE0 := W#16#0;
   SD_1_SAVE2 := W#16#0;
   SD_1_SAVE4 := W#16#0;
   SD_1_SAVE6 := W#16#0;
   SD_1_SAVE8 := W#16#0;
   HS_REQ_BYTE.rii := FALSE;
   HS_REQ_BYTE.nva := FALSE;
   HS_REQ_BYTE.ofs := FALSE;
   HS_REQ_BYTE.dir := FALSE;
   HS_REQ_BYTE.res := FALSE;
   HS_REQ_BYTE.roc := FALSE;
   HS_REQ_BYTE.nls := FALSE;
   HS_REQ_BYTE.rlo := FALSE;
   HS_RESP_BYTE.aii := FALSE;
   HS_RESP_BYTE.sns := FALSE;
   HS_RESP_BYTE.sqc := FALSE;
   HS_RESP_BYTE.ads := FALSE;
   HS_RESP_BYTE.aoc := FALSE;
   HS_RESP_BYTE.rs1 := FALSE;
   HS_RESP_BYTE.cnr := FALSE;
   HS_RESP_BYTE.rs2 := FALSE;
   HS_RESP_DSNR := B#16#0;
   HS_RESP_OFFSET := W#16#0;
   SD_1_WORD0 := W#16#0;
   SD_1_COUNT := W#16#0;
   SD_1_DBNUMMER := W#16#0;
   SD_1_DWORD6 := DW#16#0;
   SD_1_TYP := B#16#0;
   SFC_PARAM.LEN := W#16#0;
   SFC_PARAM.DB_NUMMER := W#16#0;
   SFC_PARAM.START := DW#16#0;
   BUFFER[0] := W#16#0;
   BUFFER[1] := W#16#0;
   BUFFER[2] := W#16#0;
   BUFFER[3] := W#16#0;
   BUFFER[4] := W#16#0;
   BUFFER[5] := W#16#0;
   BUFFER[6] := W#16#0;
   BUFFER[7] := W#16#0;
   BUFFER[8] := W#16#0;
   BUFFER[9] := W#16#0;
   BUFFER[10] := W#16#0;
   BUFFER[11] := W#16#0;
   BUFFER[12] := W#16#0;
   BUFFER[13] := W#16#0;
   BUFFER[14] := W#16#0;
   BUFFER[15] := W#16#0;
   BUFFER[16] := W#16#0;
   BUFFER[17] := W#16#0;
   BUFFER[18] := W#16#0;
   BUFFER[19] := W#16#0;
   BUFFER[20] := W#16#0;
   BUFFER[21] := W#16#0;
   BUFFER[22] := W#16#0;
   BUFFER[23] := W#16#0;
   BUFFER[24] := W#16#0;
   BUFFER[25] := W#16#0;
   BUFFER[26] := W#16#0;
   BUFFER[27] := W#16#0;
   BUFFER[28] := W#16#0;
   BUFFER[29] := W#16#0;
   BUFFER[30] := W#16#0;
   BUFFER[31] := W#16#0;
   BUFFER[32] := W#16#0;
   BUFFER[33] := W#16#0;
   BUFFER[34] := W#16#0;
   BUFFER[35] := W#16#0;
   BUFFER[36] := W#16#0;
   BUFFER[37] := W#16#0;
   BUFFER[38] := W#16#0;
   BUFFER[39] := W#16#0;
   BUFFER[40] := W#16#0;
   BUFFER[41] := W#16#0;
   BUFFER[42] := W#16#0;
   BUFFER[43] := W#16#0;
   BUFFER[44] := W#16#0;
   BUFFER[45] := W#16#0;
   BUFFER[46] := W#16#0;
   BUFFER[47] := W#16#0;
   BUFFER[48] := W#16#0;
   BUFFER[49] := W#16#0;
   BUFFER[50] := W#16#0;
   BUFFER[51] := W#16#0;
   BUFFER[52] := W#16#0;
   BUFFER[53] := W#16#0;
   BUFFER[54] := W#16#0;
   BUFFER[55] := W#16#0;
   BUFFER[56] := W#16#0;
   BUFFER[57] := W#16#0;
   BUFFER[58] := W#16#0;
   BUFFER[59] := W#16#0;
   BUFFER[60] := W#16#0;
   BUFFER[61] := W#16#0;
   BUFFER[62] := W#16#0;
   BUFFER[63] := W#16#0;
   BUFFER[64] := W#16#0;
   BUFFER[65] := W#16#0;
   BUFFER[66] := W#16#0;
   BUFFER[67] := W#16#0;
   BUFFER[68] := W#16#0;
   BUFFER[69] := W#16#0;
   BUFFER[70] := W#16#0;
   BUFFER[71] := W#16#0;
   BUFFER[72] := W#16#0;
   BUFFER[73] := W#16#0;
   BUFFER[74] := W#16#0;
   BUFFER[75] := W#16#0;
   BUFFER[76] := W#16#0;
   BUFFER[77] := W#16#0;
   BUFFER[78] := W#16#0;
   BUFFER[79] := W#16#0;
   BUFFER[80] := W#16#0;
   BUFFER[81] := W#16#0;
   BUFFER[82] := W#16#0;
   BUFFER[83] := W#16#0;
   BUFFER[84] := W#16#0;
   BUFFER[85] := W#16#0;
   BUFFER[86] := W#16#0;
   BUFFER[87] := W#16#0;
   BUFFER[88] := W#16#0;
   BUFFER[89] := W#16#0;
   BUFFER[90] := W#16#0;
   BUFFER[91] := W#16#0;
   BUFFER[92] := W#16#0;
   BUFFER[93] := W#16#0;
   BUFFER[94] := W#16#0;
   BUFFER[95] := W#16#0;
   BUFFER[96] := W#16#0;
   BUFFER[97] := W#16#0;
   BUFFER[98] := W#16#0;
   BUFFER[99] := W#16#0;
   BUFFER[100] := W#16#0;
   BUFFER[101] := W#16#0;
   BUFFER[102] := W#16#0;
   BUFFER[103] := W#16#0;
   BUFFER[104] := W#16#0;
   BUFFER[105] := W#16#0;
   BUFFER[106] := W#16#0;
   BUFFER[107] := W#16#0;
   BUFFER[108] := W#16#0;
   BUFFER[109] := W#16#0;
   BUFFER[110] := W#16#0;
   BUFFER[111] := W#16#0;
   BUFFER[112] := W#16#0;
   BUFFER[113] := W#16#0;
   BUFFER[114] := W#16#0;
   BUFFER[115] := W#16#0;
   BUFFER[116] := W#16#0;
   BUFFER[117] := W#16#0;
   BUFFER[118] := W#16#0;
   BUFFER[119] := W#16#0;
   REASON_FOR_CLOSE := B#16#0;
   DS_NR := B#16#0;
   PARAM_OFFSET := B#16#0;
   MAX_PUFF_LEN_SAVE := W#16#0;
   TYP_BOOL := FALSE;
   KANAL_PROBLEM := FALSE;
   KOMM_PROBLEM := FALSE;
   SEND_STARTED := FALSE;
   RECV_STARTED := FALSE;
   RESET_REQUEST := FALSE;
   RESET_EXECUTED := FALSE;
   DS200_BUSY := FALSE;
   MAX_DATA_LEN := W#16#0;
   LADDR_PTR := DW#16#0;
   FC_DATA_LEN := W#16#0;
   LADDR := W#16#0;
   SLEEP := B#16#0;
   SLEEP_EXT := B#16#0;
   ID_CLOSE := W#16#0;
   FB_KENNUNG := B#16#F1;
   RESERVE := B#16#0;
   ZUSTAND_WEICHE := B#16#2;
   SFB_AUFRUF.REQ := FALSE;
   SFB_AUFRUF.R := FALSE;
   SFB_AUFRUF.ID := W#16#14;
   SFB_AUFRUF.R_ID := DW#16#14;
   SFB_AUFRUF.DONE := FALSE;
   SFB_AUFRUF.ERROR := FALSE;
   SFB_AUFRUF.STATUS := W#16#0;
   SFB_AUFRUF.SD_1 := P#DB17.DBX 0.0 BYTE 80;
   SFB_AUFRUF.LEN := W#16#50;
   SFB_AUFRUF.INDEX := W#16#501;
   ZUSTAND_WEICHE_1 := B#16#CA;
END_DATA_BLOCK

DATA_BLOCK DB 74
TITLE =
AUTHOR : SIMATIC
FAMILY : CPU_300
VERSION : 0.0

 FB 12
BEGIN
   REQ := TRUE;
   R := FALSE;
   ID := W#16#16;
   R_ID := DW#16#110;
   DONE := FALSE;
   ERROR := FALSE;
   STATUS := W#16#0;
   SD_1 := P#DB18.DBX 0.0 BYTE 10;
   LEN := W#16#A;
   FB_ZUSTAND := B#16#0;
   REQ_SAVE := FALSE;
   R_SAVE := FALSE;
   ID_SAVE := W#16#0;
   R_ID_SAVE := DW#16#0;
   LEN_SAVE := W#16#0;
   SD_1_SAVE0 := W#16#0;
   SD_1_SAVE2 := W#16#0;
   SD_1_SAVE4 := W#16#0;
   SD_1_SAVE6 := W#16#0;
   SD_1_SAVE8 := W#16#0;
   HS_REQ_BYTE.rii := FALSE;
   HS_REQ_BYTE.nva := FALSE;
   HS_REQ_BYTE.ofs := FALSE;
   HS_REQ_BYTE.dir := FALSE;
   HS_REQ_BYTE.res := FALSE;
   HS_REQ_BYTE.roc := FALSE;
   HS_REQ_BYTE.nls := FALSE;
   HS_REQ_BYTE.rlo := FALSE;
   HS_RESP_BYTE.aii := FALSE;
   HS_RESP_BYTE.sns := FALSE;
   HS_RESP_BYTE.sqc := FALSE;
   HS_RESP_BYTE.ads := FALSE;
   HS_RESP_BYTE.aoc := FALSE;
   HS_RESP_BYTE.rs1 := FALSE;
   HS_RESP_BYTE.cnr := FALSE;
   HS_RESP_BYTE.rs2 := FALSE;
   HS_RESP_DSNR := B#16#0;
   HS_RESP_OFFSET := W#16#0;
   SD_1_WORD0 := W#16#0;
   SD_1_COUNT := W#16#0;
   SD_1_DBNUMMER := W#16#0;
   SD_1_DWORD6 := DW#16#0;
   SD_1_TYP := B#16#0;
   SFC_PARAM.LEN := W#16#0;
   SFC_PARAM.DB_NUMMER := W#16#0;
   SFC_PARAM.START := DW#16#0;
   BUFFER[0] := W#16#0;
   BUFFER[1] := W#16#0;
   BUFFER[2] := W#16#0;
   BUFFER[3] := W#16#0;
   BUFFER[4] := W#16#0;
   BUFFER[5] := W#16#0;
   BUFFER[6] := W#16#0;
   BUFFER[7] := W#16#0;
   BUFFER[8] := W#16#0;
   BUFFER[9] := W#16#0;
   BUFFER[10] := W#16#0;
   BUFFER[11] := W#16#0;
   BUFFER[12] := W#16#0;
   BUFFER[13] := W#16#0;
   BUFFER[14] := W#16#0;
   BUFFER[15] := W#16#0;
   BUFFER[16] := W#16#0;
   BUFFER[17] := W#16#0;
   BUFFER[18] := W#16#0;
   BUFFER[19] := W#16#0;
   BUFFER[20] := W#16#0;
   BUFFER[21] := W#16#0;
   BUFFER[22] := W#16#0;
   BUFFER[23] := W#16#0;
   BUFFER[24] := W#16#0;
   BUFFER[25] := W#16#0;
   BUFFER[26] := W#16#0;
   BUFFER[27] := W#16#0;
   BUFFER[28] := W#16#0;
   BUFFER[29] := W#16#0;
   BUFFER[30] := W#16#0;
   BUFFER[31] := W#16#0;
   BUFFER[32] := W#16#0;
   BUFFER[33] := W#16#0;
   BUFFER[34] := W#16#0;
   BUFFER[35] := W#16#0;
   BUFFER[36] := W#16#0;
   BUFFER[37] := W#16#0;
   BUFFER[38] := W#16#0;
   BUFFER[39] := W#16#0;
   BUFFER[40] := W#16#0;
   BUFFER[41] := W#16#0;
   BUFFER[42] := W#16#0;
   BUFFER[43] := W#16#0;
   BUFFER[44] := W#16#0;
   BUFFER[45] := W#16#0;
   BUFFER[46] := W#16#0;
   BUFFER[47] := W#16#0;
   BUFFER[48] := W#16#0;
   BUFFER[49] := W#16#0;
   BUFFER[50] := W#16#0;
   BUFFER[51] := W#16#0;
   BUFFER[52] := W#16#0;
   BUFFER[53] := W#16#0;
   BUFFER[54] := W#16#0;
   BUFFER[55] := W#16#0;
   BUFFER[56] := W#16#0;
   BUFFER[57] := W#16#0;
   BUFFER[58] := W#16#0;
   BUFFER[59] := W#16#0;
   BUFFER[60] := W#16#0;
   BUFFER[61] := W#16#0;
   BUFFER[62] := W#16#0;
   BUFFER[63] := W#16#0;
   BUFFER[64] := W#16#0;
   BUFFER[65] := W#16#0;
   BUFFER[66] := W#16#0;
   BUFFER[67] := W#16#0;
   BUFFER[68] := W#16#0;
   BUFFER[69] := W#16#0;
   BUFFER[70] := W#16#0;
   BUFFER[71] := W#16#0;
   BUFFER[72] := W#16#0;
   BUFFER[73] := W#16#0;
   BUFFER[74] := W#16#0;
   BUFFER[75] := W#16#0;
   BUFFER[76] := W#16#0;
   BUFFER[77] := W#16#0;
   BUFFER[78] := W#16#0;
   BUFFER[79] := W#16#0;
   BUFFER[80] := W#16#0;
   BUFFER[81] := W#16#0;
   BUFFER[82] := W#16#0;
   BUFFER[83] := W#16#0;
   BUFFER[84] := W#16#0;
   BUFFER[85] := W#16#0;
   BUFFER[86] := W#16#0;
   BUFFER[87] := W#16#0;
   BUFFER[88] := W#16#0;
   BUFFER[89] := W#16#0;
   BUFFER[90] := W#16#0;
   BUFFER[91] := W#16#0;
   BUFFER[92] := W#16#0;
   BUFFER[93] := W#16#0;
   BUFFER[94] := W#16#0;
   BUFFER[95] := W#16#0;
   BUFFER[96] := W#16#0;
   BUFFER[97] := W#16#0;
   BUFFER[98] := W#16#0;
   BUFFER[99] := W#16#0;
   BUFFER[100] := W#16#0;
   BUFFER[101] := W#16#0;
   BUFFER[102] := W#16#0;
   BUFFER[103] := W#16#0;
   BUFFER[104] := W#16#0;
   BUFFER[105] := W#16#0;
   BUFFER[106] := W#16#0;
   BUFFER[107] := W#16#0;
   BUFFER[108] := W#16#0;
   BUFFER[109] := W#16#0;
   BUFFER[110] := W#16#0;
   BUFFER[111] := W#16#0;
   BUFFER[112] := W#16#0;
   BUFFER[113] := W#16#0;
   BUFFER[114] := W#16#0;
   BUFFER[115] := W#16#0;
   BUFFER[116] := W#16#0;
   BUFFER[117] := W#16#0;
   BUFFER[118] := W#16#0;
   BUFFER[119] := W#16#0;
   REASON_FOR_CLOSE := B#16#0;
   DS_NR := B#16#0;
   PARAM_OFFSET := B#16#0;
   MAX_PUFF_LEN_SAVE := W#16#0;
   TYP_BOOL := FALSE;
   KANAL_PROBLEM := FALSE;
   KOMM_PROBLEM := FALSE;
   SEND_STARTED := FALSE;
   RECV_STARTED := FALSE;
   RESET_REQUEST := FALSE;
   RESET_EXECUTED := FALSE;
   DS200_BUSY := FALSE;
   MAX_DATA_LEN := W#16#0;
   LADDR_PTR := DW#16#0;
   FC_DATA_LEN := W#16#0;
   LADDR := W#16#0;
   SLEEP := B#16#0;
   SLEEP_EXT := B#16#0;
   ID_CLOSE := W#16#0;
   FB_KENNUNG := B#16#F1;
   RESERVE := B#16#0;
   ZUSTAND_WEICHE := B#16#2;
   SFB_AUFRUF.REQ := FALSE;
   SFB_AUFRUF.R := FALSE;
   SFB_AUFRUF.ID := W#16#16;
   SFB_AUFRUF.R_ID := DW#16#110;
   SFB_AUFRUF.DONE := FALSE;
   SFB_AUFRUF.ERROR := FALSE;
   SFB_AUFRUF.STATUS := W#16#0;
   SFB_AUFRUF.SD_1 := P#DB18.DBX 0.0 BYTE 10;
   SFB_AUFRUF.LEN := W#16#A;
   SFB_AUFRUF.INDEX := W#16#701;
   ZUSTAND_WEICHE_1 := B#16#CA;
END_DATA_BLOCK

DATA_BLOCK DB 81
TITLE =
AUTHOR : SIMATIC
FAMILY : CPU_300
VERSION : 0.0

 FB 13
BEGIN
   EN_R := TRUE;
   ID := W#16#3;
   R_ID := DW#16#3;
   NDR := FALSE;
   ERROR := FALSE;
   STATUS := W#16#19;
   RD_1 := P#DB1.DBX 0.0 BYTE 500;
   LEN := W#16#CC;
   FB_ZUSTAND := B#16#0;
   EN_R_SAVE := FALSE;
   ID_SAVE := W#16#0;
   R_ID_SAVE := DW#16#0;
   FC_DATA_LEN := W#16#0;
   SD_1_SAVE0 := W#16#0;
   SD_1_SAVE2 := W#16#0;
   SD_1_SAVE4 := W#16#0;
   SD_1_SAVE6 := W#16#0;
   SD_1_SAVE8 := W#16#0;
   HS_REQ_BYTE.rii := FALSE;
   HS_REQ_BYTE.nva := FALSE;
   HS_REQ_BYTE.ofs := FALSE;
   HS_REQ_BYTE.dir := FALSE;
   HS_REQ_BYTE.res := FALSE;
   HS_REQ_BYTE.roc := FALSE;
   HS_REQ_BYTE.nls := FALSE;
   HS_REQ_BYTE.rlo := FALSE;
   HS_RESP_BYTE.aii := FALSE;
   HS_RESP_BYTE.sns := FALSE;
   HS_RESP_BYTE.sqc := FALSE;
   HS_RESP_BYTE.ads := FALSE;
   HS_RESP_BYTE.aoc := FALSE;
   HS_RESP_BYTE.rs1 := FALSE;
   HS_RESP_BYTE.cnr := FALSE;
   HS_RESP_BYTE.rs2 := FALSE;
   HS_RESP_DSNR := B#16#0;
   HS_RESP_OFFSET := W#16#0;
   SD_1_WORD0 := W#16#0;
   SD_1_COUNT := W#16#0;
   SD_1_DBNUMMER := W#16#0;
   SD_1_DWORD6 := DW#16#0;
   SD_1_TYP := B#16#0;
   SFC_PARAM.LEN := W#16#0;
   SFC_PARAM.DB_NUMMER := W#16#0;
   SFC_PARAM.START := DW#16#0;
   BUFFER[0] := W#16#0;
   BUFFER[1] := W#16#0;
   BUFFER[2] := W#16#0;
   BUFFER[3] := W#16#0;
   BUFFER[4] := W#16#0;
   BUFFER[5] := W#16#0;
   BUFFER[6] := W#16#0;
   BUFFER[7] := W#16#0;
   BUFFER[8] := W#16#0;
   BUFFER[9] := W#16#0;
   BUFFER[10] := W#16#0;
   BUFFER[11] := W#16#0;
   BUFFER[12] := W#16#0;
   BUFFER[13] := W#16#0;
   BUFFER[14] := W#16#0;
   BUFFER[15] := W#16#0;
   BUFFER[16] := W#16#0;
   BUFFER[17] := W#16#0;
   BUFFER[18] := W#16#0;
   BUFFER[19] := W#16#0;
   BUFFER[20] := W#16#0;
   BUFFER[21] := W#16#0;
   BUFFER[22] := W#16#0;
   BUFFER[23] := W#16#0;
   BUFFER[24] := W#16#0;
   BUFFER[25] := W#16#0;
   BUFFER[26] := W#16#0;
   BUFFER[27] := W#16#0;
   BUFFER[28] := W#16#0;
   BUFFER[29] := W#16#0;
   BUFFER[30] := W#16#0;
   BUFFER[31] := W#16#0;
   BUFFER[32] := W#16#0;
   BUFFER[33] := W#16#0;
   BUFFER[34] := W#16#0;
   BUFFER[35] := W#16#0;
   BUFFER[36] := W#16#0;
   BUFFER[37] := W#16#0;
   BUFFER[38] := W#16#0;
   BUFFER[39] := W#16#0;
   BUFFER[40] := W#16#0;
   BUFFER[41] := W#16#0;
   BUFFER[42] := W#16#0;
   BUFFER[43] := W#16#0;
   BUFFER[44] := W#16#0;
   BUFFER[45] := W#16#0;
   BUFFER[46] := W#16#0;
   BUFFER[47] := W#16#0;
   BUFFER[48] := W#16#0;
   BUFFER[49] := W#16#0;
   BUFFER[50] := W#16#0;
   BUFFER[51] := W#16#0;
   BUFFER[52] := W#16#0;
   BUFFER[53] := W#16#0;
   BUFFER[54] := W#16#0;
   BUFFER[55] := W#16#0;
   BUFFER[56] := W#16#0;
   BUFFER[57] := W#16#0;
   BUFFER[58] := W#16#0;
   BUFFER[59] := W#16#0;
   BUFFER[60] := W#16#0;
   BUFFER[61] := W#16#0;
   BUFFER[62] := W#16#0;
   BUFFER[63] := W#16#0;
   BUFFER[64] := W#16#0;
   BUFFER[65] := W#16#0;
   BUFFER[66] := W#16#0;
   BUFFER[67] := W#16#0;
   BUFFER[68] := W#16#0;
   BUFFER[69] := W#16#0;
   BUFFER[70] := W#16#0;
   BUFFER[71] := W#16#0;
   BUFFER[72] := W#16#0;
   BUFFER[73] := W#16#0;
   BUFFER[74] := W#16#0;
   BUFFER[75] := W#16#0;
   BUFFER[76] := W#16#0;
   BUFFER[77] := W#16#0;
   BUFFER[78] := W#16#0;
   BUFFER[79] := W#16#0;
   BUFFER[80] := W#16#0;
   BUFFER[81] := W#16#0;
   BUFFER[82] := W#16#0;
   BUFFER[83] := W#16#0;
   BUFFER[84] := W#16#0;
   BUFFER[85] := W#16#0;
   BUFFER[86] := W#16#0;
   BUFFER[87] := W#16#0;
   BUFFER[88] := W#16#0;
   BUFFER[89] := W#16#0;
   BUFFER[90] := W#16#0;
   BUFFER[91] := W#16#0;
   BUFFER[92] := W#16#0;
   BUFFER[93] := W#16#0;
   BUFFER[94] := W#16#0;
   BUFFER[95] := W#16#0;
   BUFFER[96] := W#16#0;
   BUFFER[97] := W#16#0;
   BUFFER[98] := W#16#0;
   BUFFER[99] := W#16#0;
   BUFFER[100] := W#16#0;
   BUFFER[101] := W#16#0;
   BUFFER[102] := W#16#0;
   BUFFER[103] := W#16#0;
   BUFFER[104] := W#16#0;
   BUFFER[105] := W#16#0;
   BUFFER[106] := W#16#0;
   BUFFER[107] := W#16#0;
   BUFFER[108] := W#16#0;
   BUFFER[109] := W#16#0;
   BUFFER[110] := W#16#0;
   BUFFER[111] := W#16#0;
   BUFFER[112] := W#16#0;
   BUFFER[113] := W#16#0;
   BUFFER[114] := W#16#0;
   BUFFER[115] := W#16#0;
   BUFFER[116] := W#16#0;
   BUFFER[117] := W#16#0;
   BUFFER[118] := W#16#0;
   BUFFER[119] := W#16#0;
   REASON_FOR_CLOSE := B#16#0;
   DS_NR := B#16#0;
   MAX_PUFF_LEN_SAVE := W#16#0;
   TYP_BOOL := FALSE;
   KANAL_PROBLEM := FALSE;
   KOMM_PROBLEM := FALSE;
   RECV_STARTED := FALSE;
   SEND_STARTED := FALSE;
   RESET_REQUEST := FALSE;
   RESET_EXECUTED := FALSE;
   DS200_BUSY := FALSE;
   LADDR_PTR := DW#16#0;
   LADDR := W#16#0;
   ZIEL_BYTE_SAVE := B#16#0;
   BOOL_ZIEL_BAD := FALSE;
   PARAM_OFFSET := DW#16#0;
   SLEEP := B#16#0;
   SLEEP_EXT := B#16#0;
   ID_CLOSE := W#16#0;
   RUNNING_LEN := W#16#0;
   FB_KENNUNG := B#16#F2;
   RESERVE := B#16#0;
   ZUSTAND_WEICHE := B#16#2;
   SFB_AUFRUF.EN_R := TRUE;
   SFB_AUFRUF.ID := W#16#3;
   SFB_AUFRUF.R_ID := DW#16#3;
   SFB_AUFRUF.NDR := FALSE;
   SFB_AUFRUF.ERROR := FALSE;
   SFB_AUFRUF.STATUS := W#16#19;
   SFB_AUFRUF.RD_1 := P#DB1.DBX 0.0 BYTE 500;
   SFB_AUFRUF.LEN := W#16#19A;
   SFB_AUFRUF.INDEX := W#16#1;
   ZUSTAND_WEICHE_1 := B#16#CA;
END_DATA_BLOCK

DATA_BLOCK DB 82
TITLE =
AUTHOR : SIMATIC
FAMILY : CPU_300
VERSION : 0.0

 FB 13
BEGIN
   EN_R := TRUE;
   ID := W#16#4;
   R_ID := DW#16#4;
   NDR := FALSE;
   ERROR := FALSE;
   STATUS := W#16#0;
   RD_1 := P#DB12.DBX 0.0 BYTE 80;
   LEN := W#16#0;
   FB_ZUSTAND := B#16#0;
   EN_R_SAVE := FALSE;
   ID_SAVE := W#16#0;
   R_ID_SAVE := DW#16#0;
   FC_DATA_LEN := W#16#0;
   SD_1_SAVE0 := W#16#0;
   SD_1_SAVE2 := W#16#0;
   SD_1_SAVE4 := W#16#0;
   SD_1_SAVE6 := W#16#0;
   SD_1_SAVE8 := W#16#0;
   HS_REQ_BYTE.rii := FALSE;
   HS_REQ_BYTE.nva := FALSE;
   HS_REQ_BYTE.ofs := FALSE;
   HS_REQ_BYTE.dir := FALSE;
   HS_REQ_BYTE.res := FALSE;
   HS_REQ_BYTE.roc := FALSE;
   HS_REQ_BYTE.nls := FALSE;
   HS_REQ_BYTE.rlo := FALSE;
   HS_RESP_BYTE.aii := FALSE;
   HS_RESP_BYTE.sns := FALSE;
   HS_RESP_BYTE.sqc := FALSE;
   HS_RESP_BYTE.ads := FALSE;
   HS_RESP_BYTE.aoc := FALSE;
   HS_RESP_BYTE.rs1 := FALSE;
   HS_RESP_BYTE.cnr := FALSE;
   HS_RESP_BYTE.rs2 := FALSE;
   HS_RESP_DSNR := B#16#0;
   HS_RESP_OFFSET := W#16#0;
   SD_1_WORD0 := W#16#0;
   SD_1_COUNT := W#16#0;
   SD_1_DBNUMMER := W#16#0;
   SD_1_DWORD6 := DW#16#0;
   SD_1_TYP := B#16#0;
   SFC_PARAM.LEN := W#16#0;
   SFC_PARAM.DB_NUMMER := W#16#0;
   SFC_PARAM.START := DW#16#0;
   BUFFER[0] := W#16#0;
   BUFFER[1] := W#16#0;
   BUFFER[2] := W#16#0;
   BUFFER[3] := W#16#0;
   BUFFER[4] := W#16#0;
   BUFFER[5] := W#16#0;
   BUFFER[6] := W#16#0;
   BUFFER[7] := W#16#0;
   BUFFER[8] := W#16#0;
   BUFFER[9] := W#16#0;
   BUFFER[10] := W#16#0;
   BUFFER[11] := W#16#0;
   BUFFER[12] := W#16#0;
   BUFFER[13] := W#16#0;
   BUFFER[14] := W#16#0;
   BUFFER[15] := W#16#0;
   BUFFER[16] := W#16#0;
   BUFFER[17] := W#16#0;
   BUFFER[18] := W#16#0;
   BUFFER[19] := W#16#0;
   BUFFER[20] := W#16#0;
   BUFFER[21] := W#16#0;
   BUFFER[22] := W#16#0;
   BUFFER[23] := W#16#0;
   BUFFER[24] := W#16#0;
   BUFFER[25] := W#16#0;
   BUFFER[26] := W#16#0;
   BUFFER[27] := W#16#0;
   BUFFER[28] := W#16#0;
   BUFFER[29] := W#16#0;
   BUFFER[30] := W#16#0;
   BUFFER[31] := W#16#0;
   BUFFER[32] := W#16#0;
   BUFFER[33] := W#16#0;
   BUFFER[34] := W#16#0;
   BUFFER[35] := W#16#0;
   BUFFER[36] := W#16#0;
   BUFFER[37] := W#16#0;
   BUFFER[38] := W#16#0;
   BUFFER[39] := W#16#0;
   BUFFER[40] := W#16#0;
   BUFFER[41] := W#16#0;
   BUFFER[42] := W#16#0;
   BUFFER[43] := W#16#0;
   BUFFER[44] := W#16#0;
   BUFFER[45] := W#16#0;
   BUFFER[46] := W#16#0;
   BUFFER[47] := W#16#0;
   BUFFER[48] := W#16#0;
   BUFFER[49] := W#16#0;
   BUFFER[50] := W#16#0;
   BUFFER[51] := W#16#0;
   BUFFER[52] := W#16#0;
   BUFFER[53] := W#16#0;
   BUFFER[54] := W#16#0;
   BUFFER[55] := W#16#0;
   BUFFER[56] := W#16#0;
   BUFFER[57] := W#16#0;
   BUFFER[58] := W#16#0;
   BUFFER[59] := W#16#0;
   BUFFER[60] := W#16#0;
   BUFFER[61] := W#16#0;
   BUFFER[62] := W#16#0;
   BUFFER[63] := W#16#0;
   BUFFER[64] := W#16#0;
   BUFFER[65] := W#16#0;
   BUFFER[66] := W#16#0;
   BUFFER[67] := W#16#0;
   BUFFER[68] := W#16#0;
   BUFFER[69] := W#16#0;
   BUFFER[70] := W#16#0;
   BUFFER[71] := W#16#0;
   BUFFER[72] := W#16#0;
   BUFFER[73] := W#16#0;
   BUFFER[74] := W#16#0;
   BUFFER[75] := W#16#0;
   BUFFER[76] := W#16#0;
   BUFFER[77] := W#16#0;
   BUFFER[78] := W#16#0;
   BUFFER[79] := W#16#0;
   BUFFER[80] := W#16#0;
   BUFFER[81] := W#16#0;
   BUFFER[82] := W#16#0;
   BUFFER[83] := W#16#0;
   BUFFER[84] := W#16#0;
   BUFFER[85] := W#16#0;
   BUFFER[86] := W#16#0;
   BUFFER[87] := W#16#0;
   BUFFER[88] := W#16#0;
   BUFFER[89] := W#16#0;
   BUFFER[90] := W#16#0;
   BUFFER[91] := W#16#0;
   BUFFER[92] := W#16#0;
   BUFFER[93] := W#16#0;
   BUFFER[94] := W#16#0;
   BUFFER[95] := W#16#0;
   BUFFER[96] := W#16#0;
   BUFFER[97] := W#16#0;
   BUFFER[98] := W#16#0;
   BUFFER[99] := W#16#0;
   BUFFER[100] := W#16#0;
   BUFFER[101] := W#16#0;
   BUFFER[102] := W#16#0;
   BUFFER[103] := W#16#0;
   BUFFER[104] := W#16#0;
   BUFFER[105] := W#16#0;
   BUFFER[106] := W#16#0;
   BUFFER[107] := W#16#0;
   BUFFER[108] := W#16#0;
   BUFFER[109] := W#16#0;
   BUFFER[110] := W#16#0;
   BUFFER[111] := W#16#0;
   BUFFER[112] := W#16#0;
   BUFFER[113] := W#16#0;
   BUFFER[114] := W#16#0;
   BUFFER[115] := W#16#0;
   BUFFER[116] := W#16#0;
   BUFFER[117] := W#16#0;
   BUFFER[118] := W#16#0;
   BUFFER[119] := W#16#0;
   REASON_FOR_CLOSE := B#16#0;
   DS_NR := B#16#0;
   MAX_PUFF_LEN_SAVE := W#16#0;
   TYP_BOOL := FALSE;
   KANAL_PROBLEM := FALSE;
   KOMM_PROBLEM := FALSE;
   RECV_STARTED := FALSE;
   SEND_STARTED := FALSE;
   RESET_REQUEST := FALSE;
   RESET_EXECUTED := FALSE;
   DS200_BUSY := FALSE;
   LADDR_PTR := DW#16#0;
   LADDR := W#16#0;
   ZIEL_BYTE_SAVE := B#16#0;
   BOOL_ZIEL_BAD := FALSE;
   PARAM_OFFSET := DW#16#0;
   SLEEP := B#16#0;
   SLEEP_EXT := B#16#0;
   ID_CLOSE := W#16#0;
   RUNNING_LEN := W#16#0;
   FB_KENNUNG := B#16#F2;
   RESERVE := B#16#0;
   ZUSTAND_WEICHE := B#16#0;
   SFB_AUFRUF.EN_R := TRUE;
   SFB_AUFRUF.ID := W#16#4;
   SFB_AUFRUF.R_ID := DW#16#4;
   SFB_AUFRUF.NDR := TRUE;
   SFB_AUFRUF.ERROR := FALSE;
   SFB_AUFRUF.STATUS := W#16#0;
   SFB_AUFRUF.RD_1 := P#DB12.DBX 0.0 BYTE 80;
   SFB_AUFRUF.LEN := W#16#50;
   SFB_AUFRUF.INDEX := W#16#201;
   ZUSTAND_WEICHE_1 := B#16#0;
END_DATA_BLOCK

DATA_BLOCK DB 83
TITLE =
AUTHOR : SIMATIC
FAMILY : CPU_300
VERSION : 0.0

 FB 13
BEGIN
   EN_R := TRUE;
   ID := W#16#12;
   R_ID := DW#16#12;
   NDR := FALSE;
   ERROR := FALSE;
   STATUS := W#16#0;
   RD_1 := P#DB26.DBX 0.0 BYTE 20;
   LEN := W#16#0;
   FB_ZUSTAND := B#16#0;
   EN_R_SAVE := FALSE;
   ID_SAVE := W#16#0;
   R_ID_SAVE := DW#16#0;
   FC_DATA_LEN := W#16#0;
   SD_1_SAVE0 := W#16#0;
   SD_1_SAVE2 := W#16#0;
   SD_1_SAVE4 := W#16#0;
   SD_1_SAVE6 := W#16#0;
   SD_1_SAVE8 := W#16#0;
   HS_REQ_BYTE.rii := FALSE;
   HS_REQ_BYTE.nva := FALSE;
   HS_REQ_BYTE.ofs := FALSE;
   HS_REQ_BYTE.dir := FALSE;
   HS_REQ_BYTE.res := FALSE;
   HS_REQ_BYTE.roc := FALSE;
   HS_REQ_BYTE.nls := FALSE;
   HS_REQ_BYTE.rlo := FALSE;
   HS_RESP_BYTE.aii := FALSE;
   HS_RESP_BYTE.sns := FALSE;
   HS_RESP_BYTE.sqc := FALSE;
   HS_RESP_BYTE.ads := FALSE;
   HS_RESP_BYTE.aoc := FALSE;
   HS_RESP_BYTE.rs1 := FALSE;
   HS_RESP_BYTE.cnr := FALSE;
   HS_RESP_BYTE.rs2 := FALSE;
   HS_RESP_DSNR := B#16#0;
   HS_RESP_OFFSET := W#16#0;
   SD_1_WORD0 := W#16#0;
   SD_1_COUNT := W#16#0;
   SD_1_DBNUMMER := W#16#0;
   SD_1_DWORD6 := DW#16#0;
   SD_1_TYP := B#16#0;
   SFC_PARAM.LEN := W#16#0;
   SFC_PARAM.DB_NUMMER := W#16#0;
   SFC_PARAM.START := DW#16#0;
   BUFFER[0] := W#16#0;
   BUFFER[1] := W#16#0;
   BUFFER[2] := W#16#0;
   BUFFER[3] := W#16#0;
   BUFFER[4] := W#16#0;
   BUFFER[5] := W#16#0;
   BUFFER[6] := W#16#0;
   BUFFER[7] := W#16#0;
   BUFFER[8] := W#16#0;
   BUFFER[9] := W#16#0;
   BUFFER[10] := W#16#0;
   BUFFER[11] := W#16#0;
   BUFFER[12] := W#16#0;
   BUFFER[13] := W#16#0;
   BUFFER[14] := W#16#0;
   BUFFER[15] := W#16#0;
   BUFFER[16] := W#16#0;
   BUFFER[17] := W#16#0;
   BUFFER[18] := W#16#0;
   BUFFER[19] := W#16#0;
   BUFFER[20] := W#16#0;
   BUFFER[21] := W#16#0;
   BUFFER[22] := W#16#0;
   BUFFER[23] := W#16#0;
   BUFFER[24] := W#16#0;
   BUFFER[25] := W#16#0;
   BUFFER[26] := W#16#0;
   BUFFER[27] := W#16#0;
   BUFFER[28] := W#16#0;
   BUFFER[29] := W#16#0;
   BUFFER[30] := W#16#0;
   BUFFER[31] := W#16#0;
   BUFFER[32] := W#16#0;
   BUFFER[33] := W#16#0;
   BUFFER[34] := W#16#0;
   BUFFER[35] := W#16#0;
   BUFFER[36] := W#16#0;
   BUFFER[37] := W#16#0;
   BUFFER[38] := W#16#0;
   BUFFER[39] := W#16#0;
   BUFFER[40] := W#16#0;
   BUFFER[41] := W#16#0;
   BUFFER[42] := W#16#0;
   BUFFER[43] := W#16#0;
   BUFFER[44] := W#16#0;
   BUFFER[45] := W#16#0;
   BUFFER[46] := W#16#0;
   BUFFER[47] := W#16#0;
   BUFFER[48] := W#16#0;
   BUFFER[49] := W#16#0;
   BUFFER[50] := W#16#0;
   BUFFER[51] := W#16#0;
   BUFFER[52] := W#16#0;
   BUFFER[53] := W#16#0;
   BUFFER[54] := W#16#0;
   BUFFER[55] := W#16#0;
   BUFFER[56] := W#16#0;
   BUFFER[57] := W#16#0;
   BUFFER[58] := W#16#0;
   BUFFER[59] := W#16#0;
   BUFFER[60] := W#16#0;
   BUFFER[61] := W#16#0;
   BUFFER[62] := W#16#0;
   BUFFER[63] := W#16#0;
   BUFFER[64] := W#16#0;
   BUFFER[65] := W#16#0;
   BUFFER[66] := W#16#0;
   BUFFER[67] := W#16#0;
   BUFFER[68] := W#16#0;
   BUFFER[69] := W#16#0;
   BUFFER[70] := W#16#0;
   BUFFER[71] := W#16#0;
   BUFFER[72] := W#16#0;
   BUFFER[73] := W#16#0;
   BUFFER[74] := W#16#0;
   BUFFER[75] := W#16#0;
   BUFFER[76] := W#16#0;
   BUFFER[77] := W#16#0;
   BUFFER[78] := W#16#0;
   BUFFER[79] := W#16#0;
   BUFFER[80] := W#16#0;
   BUFFER[81] := W#16#0;
   BUFFER[82] := W#16#0;
   BUFFER[83] := W#16#0;
   BUFFER[84] := W#16#0;
   BUFFER[85] := W#16#0;
   BUFFER[86] := W#16#0;
   BUFFER[87] := W#16#0;
   BUFFER[88] := W#16#0;
   BUFFER[89] := W#16#0;
   BUFFER[90] := W#16#0;
   BUFFER[91] := W#16#0;
   BUFFER[92] := W#16#0;
   BUFFER[93] := W#16#0;
   BUFFER[94] := W#16#0;
   BUFFER[95] := W#16#0;
   BUFFER[96] := W#16#0;
   BUFFER[97] := W#16#0;
   BUFFER[98] := W#16#0;
   BUFFER[99] := W#16#0;
   BUFFER[100] := W#16#0;
   BUFFER[101] := W#16#0;
   BUFFER[102] := W#16#0;
   BUFFER[103] := W#16#0;
   BUFFER[104] := W#16#0;
   BUFFER[105] := W#16#0;
   BUFFER[106] := W#16#0;
   BUFFER[107] := W#16#0;
   BUFFER[108] := W#16#0;
   BUFFER[109] := W#16#0;
   BUFFER[110] := W#16#0;
   BUFFER[111] := W#16#0;
   BUFFER[112] := W#16#0;
   BUFFER[113] := W#16#0;
   BUFFER[114] := W#16#0;
   BUFFER[115] := W#16#0;
   BUFFER[116] := W#16#0;
   BUFFER[117] := W#16#0;
   BUFFER[118] := W#16#0;
   BUFFER[119] := W#16#0;
   REASON_FOR_CLOSE := B#16#0;
   DS_NR := B#16#0;
   MAX_PUFF_LEN_SAVE := W#16#0;
   TYP_BOOL := FALSE;
   KANAL_PROBLEM := FALSE;
   KOMM_PROBLEM := FALSE;
   RECV_STARTED := FALSE;
   SEND_STARTED := FALSE;
   RESET_REQUEST := FALSE;
   RESET_EXECUTED := FALSE;
   DS200_BUSY := FALSE;
   LADDR_PTR := DW#16#0;
   LADDR := W#16#0;
   ZIEL_BYTE_SAVE := B#16#0;
   BOOL_ZIEL_BAD := FALSE;
   PARAM_OFFSET := DW#16#0;
   SLEEP := B#16#0;
   SLEEP_EXT := B#16#0;
   ID_CLOSE := W#16#0;
   RUNNING_LEN := W#16#0;
   FB_KENNUNG := B#16#F2;
   RESERVE := B#16#0;
   ZUSTAND_WEICHE := B#16#2;
   SFB_AUFRUF.EN_R := TRUE;
   SFB_AUFRUF.ID := W#16#12;
   SFB_AUFRUF.R_ID := DW#16#12;
   SFB_AUFRUF.NDR := FALSE;
   SFB_AUFRUF.ERROR := FALSE;
   SFB_AUFRUF.STATUS := W#16#0;
   SFB_AUFRUF.RD_1 := P#DB26.DBX 0.0 BYTE 20;
   SFB_AUFRUF.LEN := W#16#0;
   SFB_AUFRUF.INDEX := W#16#401;
   ZUSTAND_WEICHE_1 := B#16#CA;
END_DATA_BLOCK

DATA_BLOCK DB 84
TITLE =
AUTHOR : SIMATIC
FAMILY : CPU_300
VERSION : 0.0

 FB 13
BEGIN
   EN_R := TRUE;
   ID := W#16#14;
   R_ID := DW#16#14;
   NDR := FALSE;
   ERROR := FALSE;
   STATUS := W#16#0;
   RD_1 := P#DB27.DBX 0.0 BYTE 80;
   LEN := W#16#0;
   FB_ZUSTAND := B#16#0;
   EN_R_SAVE := FALSE;
   ID_SAVE := W#16#0;
   R_ID_SAVE := DW#16#0;
   FC_DATA_LEN := W#16#0;
   SD_1_SAVE0 := W#16#0;
   SD_1_SAVE2 := W#16#0;
   SD_1_SAVE4 := W#16#0;
   SD_1_SAVE6 := W#16#0;
   SD_1_SAVE8 := W#16#0;
   HS_REQ_BYTE.rii := FALSE;
   HS_REQ_BYTE.nva := FALSE;
   HS_REQ_BYTE.ofs := FALSE;
   HS_REQ_BYTE.dir := FALSE;
   HS_REQ_BYTE.res := FALSE;
   HS_REQ_BYTE.roc := FALSE;
   HS_REQ_BYTE.nls := FALSE;
   HS_REQ_BYTE.rlo := FALSE;
   HS_RESP_BYTE.aii := FALSE;
   HS_RESP_BYTE.sns := FALSE;
   HS_RESP_BYTE.sqc := FALSE;
   HS_RESP_BYTE.ads := FALSE;
   HS_RESP_BYTE.aoc := FALSE;
   HS_RESP_BYTE.rs1 := FALSE;
   HS_RESP_BYTE.cnr := FALSE;
   HS_RESP_BYTE.rs2 := FALSE;
   HS_RESP_DSNR := B#16#0;
   HS_RESP_OFFSET := W#16#0;
   SD_1_WORD0 := W#16#0;
   SD_1_COUNT := W#16#0;
   SD_1_DBNUMMER := W#16#0;
   SD_1_DWORD6 := DW#16#0;
   SD_1_TYP := B#16#0;
   SFC_PARAM.LEN := W#16#0;
   SFC_PARAM.DB_NUMMER := W#16#0;
   SFC_PARAM.START := DW#16#0;
   BUFFER[0] := W#16#0;
   BUFFER[1] := W#16#0;
   BUFFER[2] := W#16#0;
   BUFFER[3] := W#16#0;
   BUFFER[4] := W#16#0;
   BUFFER[5] := W#16#0;
   BUFFER[6] := W#16#0;
   BUFFER[7] := W#16#0;
   BUFFER[8] := W#16#0;
   BUFFER[9] := W#16#0;
   BUFFER[10] := W#16#0;
   BUFFER[11] := W#16#0;
   BUFFER[12] := W#16#0;
   BUFFER[13] := W#16#0;
   BUFFER[14] := W#16#0;
   BUFFER[15] := W#16#0;
   BUFFER[16] := W#16#0;
   BUFFER[17] := W#16#0;
   BUFFER[18] := W#16#0;
   BUFFER[19] := W#16#0;
   BUFFER[20] := W#16#0;
   BUFFER[21] := W#16#0;
   BUFFER[22] := W#16#0;
   BUFFER[23] := W#16#0;
   BUFFER[24] := W#16#0;
   BUFFER[25] := W#16#0;
   BUFFER[26] := W#16#0;
   BUFFER[27] := W#16#0;
   BUFFER[28] := W#16#0;
   BUFFER[29] := W#16#0;
   BUFFER[30] := W#16#0;
   BUFFER[31] := W#16#0;
   BUFFER[32] := W#16#0;
   BUFFER[33] := W#16#0;
   BUFFER[34] := W#16#0;
   BUFFER[35] := W#16#0;
   BUFFER[36] := W#16#0;
   BUFFER[37] := W#16#0;
   BUFFER[38] := W#16#0;
   BUFFER[39] := W#16#0;
   BUFFER[40] := W#16#0;
   BUFFER[41] := W#16#0;
   BUFFER[42] := W#16#0;
   BUFFER[43] := W#16#0;
   BUFFER[44] := W#16#0;
   BUFFER[45] := W#16#0;
   BUFFER[46] := W#16#0;
   BUFFER[47] := W#16#0;
   BUFFER[48] := W#16#0;
   BUFFER[49] := W#16#0;
   BUFFER[50] := W#16#0;
   BUFFER[51] := W#16#0;
   BUFFER[52] := W#16#0;
   BUFFER[53] := W#16#0;
   BUFFER[54] := W#16#0;
   BUFFER[55] := W#16#0;
   BUFFER[56] := W#16#0;
   BUFFER[57] := W#16#0;
   BUFFER[58] := W#16#0;
   BUFFER[59] := W#16#0;
   BUFFER[60] := W#16#0;
   BUFFER[61] := W#16#0;
   BUFFER[62] := W#16#0;
   BUFFER[63] := W#16#0;
   BUFFER[64] := W#16#0;
   BUFFER[65] := W#16#0;
   BUFFER[66] := W#16#0;
   BUFFER[67] := W#16#0;
   BUFFER[68] := W#16#0;
   BUFFER[69] := W#16#0;
   BUFFER[70] := W#16#0;
   BUFFER[71] := W#16#0;
   BUFFER[72] := W#16#0;
   BUFFER[73] := W#16#0;
   BUFFER[74] := W#16#0;
   BUFFER[75] := W#16#0;
   BUFFER[76] := W#16#0;
   BUFFER[77] := W#16#0;
   BUFFER[78] := W#16#0;
   BUFFER[79] := W#16#0;
   BUFFER[80] := W#16#0;
   BUFFER[81] := W#16#0;
   BUFFER[82] := W#16#0;
   BUFFER[83] := W#16#0;
   BUFFER[84] := W#16#0;
   BUFFER[85] := W#16#0;
   BUFFER[86] := W#16#0;
   BUFFER[87] := W#16#0;
   BUFFER[88] := W#16#0;
   BUFFER[89] := W#16#0;
   BUFFER[90] := W#16#0;
   BUFFER[91] := W#16#0;
   BUFFER[92] := W#16#0;
   BUFFER[93] := W#16#0;
   BUFFER[94] := W#16#0;
   BUFFER[95] := W#16#0;
   BUFFER[96] := W#16#0;
   BUFFER[97] := W#16#0;
   BUFFER[98] := W#16#0;
   BUFFER[99] := W#16#0;
   BUFFER[100] := W#16#0;
   BUFFER[101] := W#16#0;
   BUFFER[102] := W#16#0;
   BUFFER[103] := W#16#0;
   BUFFER[104] := W#16#0;
   BUFFER[105] := W#16#0;
   BUFFER[106] := W#16#0;
   BUFFER[107] := W#16#0;
   BUFFER[108] := W#16#0;
   BUFFER[109] := W#16#0;
   BUFFER[110] := W#16#0;
   BUFFER[111] := W#16#0;
   BUFFER[112] := W#16#0;
   BUFFER[113] := W#16#0;
   BUFFER[114] := W#16#0;
   BUFFER[115] := W#16#0;
   BUFFER[116] := W#16#0;
   BUFFER[117] := W#16#0;
   BUFFER[118] := W#16#0;
   BUFFER[119] := W#16#0;
   REASON_FOR_CLOSE := B#16#0;
   DS_NR := B#16#0;
   MAX_PUFF_LEN_SAVE := W#16#0;
   TYP_BOOL := FALSE;
   KANAL_PROBLEM := FALSE;
   KOMM_PROBLEM := FALSE;
   RECV_STARTED := FALSE;
   SEND_STARTED := FALSE;
   RESET_REQUEST := FALSE;
   RESET_EXECUTED := FALSE;
   DS200_BUSY := FALSE;
   LADDR_PTR := DW#16#0;
   LADDR := W#16#0;
   ZIEL_BYTE_SAVE := B#16#0;
   BOOL_ZIEL_BAD := FALSE;
   PARAM_OFFSET := DW#16#0;
   SLEEP := B#16#0;
   SLEEP_EXT := B#16#0;
   ID_CLOSE := W#16#0;
   RUNNING_LEN := W#16#0;
   FB_KENNUNG := B#16#F2;
   RESERVE := B#16#0;
   ZUSTAND_WEICHE := B#16#2;
   SFB_AUFRUF.EN_R := TRUE;
   SFB_AUFRUF.ID := W#16#14;
   SFB_AUFRUF.R_ID := DW#16#14;
   SFB_AUFRUF.NDR := FALSE;
   SFB_AUFRUF.ERROR := FALSE;
   SFB_AUFRUF.STATUS := W#16#0;
   SFB_AUFRUF.RD_1 := P#DB27.DBX 0.0 BYTE 80;
   SFB_AUFRUF.LEN := W#16#0;
   SFB_AUFRUF.INDEX := W#16#601;
   ZUSTAND_WEICHE_1 := B#16#CA;
END_DATA_BLOCK

DATA_BLOCK DB 85
TITLE =
AUTHOR : SIMATIC
FAMILY : CPU_300
VERSION : 0.0

